KUKA KRL program: MyProgram_112().src

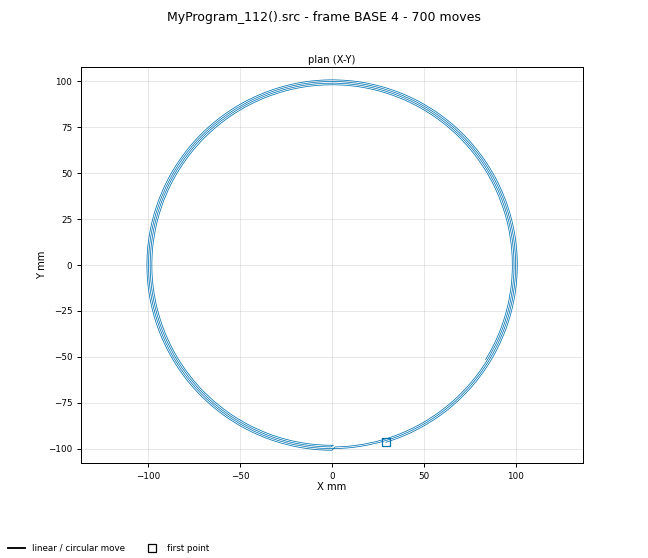
[picture p0: tool path of MyProgram_112().src in frame BASE 4, 700 of 700 moves have a stored position in this frame; points joined in program order, loops and branches not executed]
&ACCESS RVP
&REL 1
&PARAM TEMPLATE = C:\KRC\Roboter\Template\vorgabe
&PARAM EDITMASK = *
DEF MyProgram_112()
; ---- Setting reference (Base) ----
$BASE = BASE_DATA[4]

; --------------------------
; ---- Setting tool (TCP) ----
$TOOL = TOOL_DATA[3]
; --------------------------

$VEL.CP = VEL_APROX_PRINT
Startdeposition()
$VEL.CP = VEL_PRINT
LIN {X 29.2721,Y -96.4972,Z 98,A -76.9707,B 24.9412,C -1.7725,E1 25.0477,E2 162.427} C_DIS
LIN {X 31.6614,Y -95.7396,Z 98,A -75.5501,B 24.941,C -1.7741,E1 25.0514,E2 161.0052} C_DIS
LIN {X 34.0983,Y -94.8985,Z 98,A -74.1594,B 24.941,C -1.7731,E1 25.0551,E2 159.6197} C_DIS
LIN {X 36.321,Y -94.0708,Z 98,A -72.7622,B 24.9408,C -1.7768,E1 25.0587,E2 158.2167} C_DIS
LIN {X 38.5895,Y -93.1634,Z 98,A -71.3458,B 24.9406,C -1.7799,E1 25.0624,E2 156.7962} C_DIS
LIN {X 40.8931,Y -92.1753,Z 98,A -69.8287,B 24.9402,C -1.7857,E1 25.0663,E2 155.269} C_DIS
LIN {X 43.7262,Y -90.8637,Z 98,A -68.0842,B 24.9402,C -1.7874,E1 25.0707,E2 153.525} C_DIS
LIN {X 46.4684,Y -89.4942,Z 98,A -66.439,B 24.9402,C -1.7865,E1 25.0748,E2 151.8866} C_DIS
LIN {X 48.6507,Y -88.3269,Z 98,A -65.038,B 24.94,C -1.7887,E1 25.0782,E2 150.4844} C_DIS
LIN {X 50.7765,Y -87.1224,Z 98,A -63.6258,B 24.9398,C -1.7922,E1 25.0817,E2 149.0682} C_DIS
LIN {X 52.9261,Y -85.8333,Z 98,A -62.2366,B 24.9398,C -1.7935,E1 25.085,E2 147.6803} C_DIS
LIN {X 54.9902,Y -84.526,Z 98,A -60.7105,B 24.9392,C -1.8017,E1 25.0886,E2 146.1398} C_DIS
LIN {X 57.048,Y -83.151,Z 98,A -59.4381,B 24.9393,C -1.7991,E1 25.0915,E2 144.8777} C_DIS
LIN {X 59.0714,Y -81.7259,Z 98,A -57.9396,B 24.9389,C -1.8057,E1 25.0949,E2 143.3689} C_DIS
LIN {X 61.0593,Y -80.2516,Z 98,A -56.6545,B 24.939,C -1.8038,E1 25.0978,E2 142.0928} C_DIS
LIN {X 63.0104,Y -78.729,Z 98,A -55.2547,B 24.9388,C -1.8066,E1 25.1009,E2 140.6917} C_DIS
LIN {X 64.9235,Y -77.1589,Z 98,A -53.7285,B 24.9383,C -1.8146,E1 25.1042,E2 139.1525} C_DIS
LIN {X 66.8211,Y -75.5213,Z 98,A -52.4544,B 24.9385,C -1.8118,E1 25.1068,E2 137.8899} C_DIS
LIN {X 68.6313,Y -73.8803,Z 98,A -51.041,B 24.9382,C -1.8161,E1 25.1097,E2 136.4722} C_DIS
LIN {X 70.4463,Y -72.1516,Z 98,A -49.6565,B 24.9381,C -1.8179,E1 25.1125,E2 135.0891} C_DIS
LIN {X 72.1738,Y -70.4238,Z 98,A -48.2431,B 24.9378,C -1.8224,E1 25.1153,E2 133.6713} C_DIS
LIN {X 74.0767,Y -68.4173,Z 98,A -46.8469,B 24.938,C -1.8192,E1 25.1179,E2 132.2886} C_DIS
LIN {X 75.5424,Y -66.7975,Z 98,A -45.446,B 24.9373,C -1.8289,E1 25.1206,E2 130.8712} C_DIS
LIN {X 77.1791,Y -64.8992,Z 98,A -44.0458,B 24.9371,C -1.8316,E1 25.1231,E2 129.4709} C_DIS
LIN {X 78.7486,Y -62.9856,Z 98,A -42.6477,B 24.9369,C -1.835,E1 25.1256,E2 128.0713} C_DIS
LIN {X 80.2706,Y -61.034,Z 98,A -41.2495,B 24.9366,C -1.8385,E1 25.1279,E2 126.6716} C_DIS
LIN {X 81.7259,Y -59.0714,Z 98,A -39.8536,B 24.9364,C -1.8426,E1 25.1303,E2 125.2726} C_DIS
LIN {X 83.1687,Y -57.0218,Z 98,A -38.454,B 24.9362,C -1.8455,E1 25.1325,E2 123.873} C_DIS
LIN {X 84.526,Y -54.9902,Z 98,A -37.0742,B 24.9359,C -1.8491,E1 25.1346,E2 122.4917} C_DIS
LIN {X 85.8501,Y -52.8992,Z 98,A -35.6606,B 24.9356,C -1.8534,E1 25.1367,E2 121.0751} C_DIS
LIN {X 87.1224,Y -50.7765,Z 98,A -34.2789,B 24.9354,C -1.8565,E1 25.1387,E2 119.6932} C_DIS
LIN {X 88.3423,Y -48.6231,Z 98,A -32.8817,B 24.9351,C -1.8602,E1 25.1406,E2 118.2945} C_DIS
LIN {X 89.5233,Y -46.4122,Z 98,A -31.3317,B 24.9345,C -1.8696,E1 25.1426,E2 116.7305} C_DIS
LIN {X 90.7517,Y -43.9591,Z 98,A -30.0524,B 24.935,C -1.8628,E1 25.1441,E2 115.474} C_DIS
LIN {X 91.6799,Y -41.9925,Z 98,A -28.6902,B 24.9343,C -1.8717,E1 25.1458,E2 114.0982} C_DIS
LIN {X 92.6951,Y -39.7007,Z 98,A -27.2754,B 24.9341,C -1.8757,E1 25.1473,E2 112.6818} C_DIS
LIN {X 93.6299,Y -37.4434,Z 98,A -25.8803,B 24.9337,C -1.8802,E1 25.1488,E2 111.2837} C_DIS
LIN {X 94.5206,Y -35.1343,Z 98,A -24.4705,B 24.9334,C -1.8847,E1 25.1502,E2 109.8712} C_DIS
LIN {X 95.3544,Y -32.8041,Z 98,A -23.0868,B 24.9332,C -1.8882,E1 25.1515,E2 108.487} C_DIS
LIN {X 96.1401,Y -30.4239,Z 98,A -21.7045,B 24.933,C -1.8909,E1 25.1527,E2 107.106} C_DIS
LIN {X 96.8491,Y -28.0857,Z 98,A -20.3095,B 24.9326,C -1.8956,E1 25.1538,E2 105.708} C_DIS
LIN {X 97.8173,Y -24.5019,Z 98,A -18.2145,B 24.9322,C -1.9017,E1 25.1553,E2 103.6107} C_DIS
LIN {X 98.3891,Y -22.094,Z 98,A -16.8179,B 24.9319,C -1.9058,E1 25.1561,E2 102.2126} C_DIS
LIN {X 98.9077,Y -19.6417,Z 98,A -15.4202,B 24.9317,C -1.9092,E1 25.1569,E2 100.8148} C_DIS
LIN {X 99.3547,Y -17.2397,Z 98,A -14.009,B 24.9313,C -1.9146,E1 25.1576,E2 99.3992} C_DIS
LIN {X 99.7479,Y -14.7962,Z 98,A -12.4664,B 24.9305,C -1.9248,E1 25.1583,E2 97.8418} C_DIS
LIN {X 100.2282,Y -11.0833,Z 98,A -10.516,B 24.9305,C -1.9244,E1 25.1589,E2 95.9039} C_DIS
LIN {X 100.47,Y -8.6202,Z 98,A -9.1359,B 24.9303,C -1.9278,E1 25.1593,E2 94.5238} C_DIS
LIN {X 100.6495,Y -6.1835,Z 98,A -7.7249,B 24.9299,C -1.9332,E1 25.1595,E2 93.1083} C_DIS
LIN {X 100.7719,Y -3.68,Z 98,A -6.3269,B 24.9297,C -1.9368,E1 25.1597,E2 91.7103} C_DIS
LIN {X 100.833,Y -1.0408,Z 98,A -4.8838,B 24.9295,C -1.9393,E1 25.1597,E2 90.2699} C_DIS
LIN {X 100.8317,Y 1.2374,Z 98,A -3.5517,B 24.9291,C -1.945,E1 25.1597,E2 88.9323} C_DIS
LIN {X 100.7178,Y 4.9479,Z 98,A -1.4406,B 24.9286,C -1.9518,E1 25.1595,E2 86.8176} C_DIS
LIN {X 100.5661,Y 7.4182,Z 98,A -0.0444,B 24.9283,C -1.9559,E1 25.1593,E2 85.42} C_DIS
LIN {X 100.3193,Y 10.2126,Z 98,A 1.3731,B 24.9284,C -1.9538,E1 25.1589,E2 84.0159} C_DIS
LIN {X 100.0809,Y 12.3438,Z 98,A 2.749,B 24.9277,C -1.9641,E1 25.1585,E2 82.6238} C_DIS
LIN {X 99.743,Y 14.8274,Z 98,A 4.1309,B 24.9275,C -1.9669,E1 25.1579,E2 81.2435} C_DIS
LIN {X 99.3239,Y 17.4113,Z 98,A 5.759,B 24.9267,C -1.9773,E1 25.1571,E2 79.6004} C_DIS
LIN {X 98.7221,Y 20.5475,Z 98,A 7.481,B 24.9266,C -1.9792,E1 25.1562,E2 77.884} C_DIS
LIN {X 98.1031,Y 23.3304,Z 98,A 9.0196,B 24.9264,C -1.9809,E1 25.1552,E2 76.3504} C_DIS
LIN {X 97.501,Y 25.731,Z 98,A 10.4326,B 24.9261,C -1.9855,E1 25.1543,E2 74.9346} C_DIS
LIN {X 96.8491,Y 28.0857,Z 98,A 11.9161,B 24.9255,C -1.9936,E1 25.1531,E2 73.4406} C_DIS
LIN {X 96.0806,Y 30.6089,Z 98,A 13.2351,B 24.9257,C -1.9908,E1 25.152,E2 72.1357} C_DIS
LIN {X 95.3544,Y 32.8041,Z 98,A 14.6225,B 24.9252,C -1.9977,E1 25.1508,E2 70.7398} C_DIS
LIN {X 94.5094,Y 35.1638,Z 98,A 16.0209,B 24.9249,C -2.0008,E1 25.1494,E2 69.3418} C_DIS
LIN {X 93.4675,Y 37.8423,Z 98,A 17.4449,B 24.9252,C -1.9972,E1 25.148,E2 67.9342} C_DIS
LIN {X 92.6702,Y 39.7589,Z 98,A 18.7998,B 24.9244,C -2.0076,E1 25.1465,E2 66.5621} C_DIS
LIN {X 91.6665,Y 42.0211,Z 98,A 20.2138,B 24.9241,C -2.012,E1 25.1449,E2 65.1456} C_DIS
LIN {X 90.6217,Y 44.2297,Z 98,A 21.7975,B 24.9232,C -2.0238,E1 25.1429,E2 63.5425} C_DIS
LIN {X 88.9323,Y 47.5353,Z 98,A 23.6902,B 24.9234,C -2.0208,E1 25.1405,E2 61.6667} C_DIS
LIN {X 87.7232,Y 49.7309,Z 98,A 25.27,B 24.9227,C -2.031,E1 25.1383,E2 60.0712} C_DIS
LIN {X 85.8333,Y 52.9261,Z 98,A 27.2035,B 24.9227,C -2.0295,E1 25.1356,E2 58.1511} C_DIS
LIN {X 84.5086,Y 55.0166,Z 98,A 28.585,B 24.9226,C -2.0322,E1 25.1335,E2 56.7702} C_DIS
LIN {X 83.151,Y 57.048,Z 98,A 29.9824,B 24.9223,C -2.0361,E1 25.1313,E2 55.3705} C_DIS
LIN {X 81.7259,Y 59.0714,Z 98,A 31.3809,B 24.922,C -2.0393,E1 25.129,E2 53.9713} C_DIS
LIN {X 80.2323,Y 61.0843,Z 98,A 32.781,B 24.9218,C -2.0418,E1 25.1267,E2 52.5718} C_DIS
LIN {X 78.729,Y 63.0104,Z 98,A 34.1786,B 24.9215,C -2.0455,E1 25.1242,E2 51.1721} C_DIS
LIN {X 77.1384,Y 64.9476,Z 98,A 35.6387,B 24.9212,C -2.0503,E1 25.1216,E2 49.7074} C_DIS
LIN {X 75.5424,Y 66.7975,Z 98,A 36.9774,B 24.9211,C -2.0515,E1 25.1192,E2 48.3719} C_DIS
LIN {X 73.8587,Y 68.6543,Z 98,A 38.3941,B 24.9209,C -2.0544,E1 25.1165,E2 46.9546} C_DIS
LIN {X 72.1516,Y 70.4463,Z 98,A 39.7773,B 24.9207,C -2.0565,E1 25.1138,E2 45.5723} C_DIS
LIN {X 70.401,Y 72.1957,Z 98,A 41.1938,B 24.9204,C -2.0599,E1 25.111,E2 44.1537} C_DIS
LIN {X 68.2383,Y 74.2409,Z 98,A 42.8629,B 24.9202,C -2.0625,E1 25.1076,E2 42.4853} C_DIS
LIN {X 65.8414,Y 76.3769,Z 98,A 44.7266,B 24.9198,C -2.0677,E1 25.1037,E2 40.6168} C_DIS
LIN {X 63.9472,Y 77.9697,Z 98,A 46.0779,B 24.9198,C -2.0682,E1 25.1008,E2 39.2695} C_DIS
LIN {X 62.0395,Y 79.4963,Z 98,A 47.493,B 24.9195,C -2.0718,E1 25.0977,E2 37.8511} C_DIS
LIN {X 60.0699,Y 80.9949,Z 98,A 48.8783,B 24.9194,C -2.0734,E1 25.0946,E2 36.4669} C_DIS
LIN {X 58.0641,Y 82.4447,Z 98,A 50.2792,B 24.9192,C -2.0756,E1 25.0914,E2 35.0657} C_DIS
LIN {X 56.0233,Y 83.8448,Z 98,A 51.6803,B 24.919,C -2.0777,E1 25.0881,E2 33.6643} C_DIS
LIN {X 53.9488,Y 85.1944,Z 98,A 53.0977,B 24.9188,C -2.0804,E1 25.0848,E2 32.2452} C_DIS
LIN {X 51.5639,Y 86.657,Z 98,A 54.5198,B 24.9192,C -2.0763,E1 25.0814,E2 30.8373} C_DIS
LIN {X 49.6759,Y 87.7544,Z 98,A 55.9032,B 24.9186,C -2.0836,E1 25.0781,E2 29.4408} C_DIS
LIN {X 47.5073,Y 88.947,Z 98,A 57.289,B 24.9186,C -2.0847,E1 25.0747,E2 28.0563} C_DIS
LIN {X 45.1019,Y 90.1894,Z 98,A 58.8834,B 24.9182,C -2.0888,E1 25.0707,E2 26.4565} C_DIS
LIN {X 41.9636,Y 91.6928,Z 98,A 60.795,B 24.9182,C -2.0886,E1 25.0659,E2 24.5503} C_DIS
LIN {X 39.7299,Y 92.6828,Z 98,A 62.1964,B 24.918,C -2.0907,E1 25.0623,E2 23.1475} C_DIS
LIN {X 37.4434,Y 93.6299,Z 98,A 63.618,B 24.9179,C -2.0927,E1 25.0586,E2 21.7243} C_DIS
LIN {X 33.9717,Y 94.9446,Z 98,A 65.7047,B 24.9178,C -2.0938,E1 25.0531,E2 19.6394} C_DIS
LIN {X 31.3215,Y 95.85,Z 98,A 67.1448,B 24.9181,C -2.0894,E1 25.0494,E2 18.2124} C_DIS
LIN {X 28.9746,Y 96.5854,Z 98,A 68.7109,B 24.9175,C -2.0969,E1 25.0451,E2 16.6315} C_DIS
LIN {X 25.6699,Y 97.5171,Z 98,A 70.6199,B 24.9175,C -2.0966,E1 25.04,E2 14.7264} C_DIS
LIN {X 23.2997,Y 98.1106,Z 98,A 72.0231,B 24.9175,C -2.0979,E1 25.0362,E2 13.322} C_DIS
LIN {X 20.854,Y 98.6592,Z 98,A 73.4458,B 24.9175,C -2.0986,E1 25.0323,E2 11.8996} C_DIS
LIN {X 18.4576,Y 99.1357,Z 98,A 74.8488,B 24.9173,C -2.0997,E1 25.0285,E2 10.4955} C_DIS
LIN {X 15.9879,Y 99.5636,Z 98,A 76.2394,B 24.9173,C -2.0989,E1 25.0246,E2 9.1082} C_DIS
LIN {X 13.5397,Y 99.926,Z 98,A 77.6611,B 24.9173,C -2.0999,E1 25.0207,E2 7.6855} C_DIS
LIN {X 11.0833,Y 100.2282,Z 98,A 79.0669,B 24.9173,C -2.1001,E1 25.0168,E2 6.2802} C_DIS
LIN {X 8.2393,Y 100.5004,Z 98,A 80.4739,B 24.9179,C -2.0922,E1 25.013,E2 4.8927} C_DIS
LIN {X 6.1835,Y 100.6495,Z 98,A 81.8774,B 24.9172,C -2.1009,E1 25.009,E2 3.4694} C_DIS
LIN {X 3.68,Y 100.7719,Z 98,A 83.3917,B 24.917,C -2.1041,E1 25.0047,E2 1.9478} C_DIS
LIN {X 1.2375,Y 100.8317,Z 98,A 84.6904,B 24.9172,C -2.1006,E1 25.0011,E2 0.6576} C_DIS
LIN {X -1.2375,Y 100.8317,Z 98,A 86.155,B 24.9172,C -2.1025,E1 24.997,E2 -0.8114} C_DIS
LIN {X -3.7432,Y 100.7696,Z 98,A 87.4895,B 24.9174,C -2.0987,E1 24.9933,E2 -2.1373} C_DIS
LIN {X -6.2151,Y 100.6474,Z 98,A 88.8969,B 24.9174,C -2.0982,E1 24.9894,E2 -3.5439} C_DIS
LIN {X -8.7058,Y 100.4624,Z 98,A 90.4498,B 24.9171,C -2.1025,E1 24.9851,E2 -5.1076} C_DIS
LIN {X -11.1147,Y 100.2249,Z 98,A 91.7112,B 24.9175,C -2.0976,E1 24.9816,E2 -6.3581} C_DIS
LIN {X -13.8731,Y 99.879,Z 98,A 93.327,B 24.9175,C -2.098,E1 24.9771,E2 -7.976} C_DIS
LIN {X -17.2708,Y 99.3491,Z 98,A 95.2333,B 24.9177,C -2.0948,E1 24.9719,E2 -9.8766} C_DIS
LIN {X -19.7037,Y 98.8953,Z 98,A 96.8487,B 24.9172,C -2.1013,E1 24.9674,E2 -11.5092} C_DIS
LIN {X -23.3304,Y 98.1031,Z 98,A 98.7557,B 24.9179,C -2.0921,E1 24.9623,E2 -13.3967} C_DIS
LIN {X -25.731,Y 97.501,Z 98,A 100.1813,B 24.9179,C -2.0914,E1 24.9584,E2 -14.8227} C_DIS
LIN {X -28.116,Y 96.8401,Z 98,A 101.5743,B 24.9181,C -2.0894,E1 24.9547,E2 -16.2133} C_DIS
LIN {X -30.4541,Y 96.1307,Z 98,A 102.999,B 24.9181,C -2.0891,E1 24.9509,E2 -17.6398} C_DIS
LIN {X -32.8339,Y 95.3439,Z 98,A 104.4107,B 24.9183,C -2.087,E1 24.9471,E2 -19.0491} C_DIS
LIN {X -35.1343,Y 94.5206,Z 98,A 105.9422,B 24.9181,C -2.0903,E1 24.9431,E2 -20.5916} C_DIS
LIN {X -37.4434,Y 93.6299,Z 98,A 107.2295,B 24.9185,C -2.0841,E1 24.9398,E2 -21.867} C_DIS
LIN {X -39.7589,Y 92.6702,Z 98,A 108.6255,B 24.9188,C -2.0811,E1 24.9362,E2 -23.2589} C_DIS
LIN {X -41.9925,Y 91.6799,Z 98,A 110.0512,B 24.9188,C -2.0803,E1 24.9326,E2 -24.6863} C_DIS
LIN {X -44.2581,Y 90.6077,Z 98,A 111.5825,B 24.9188,C -2.0819,E1 24.9287,E2 -26.2253} C_DIS
LIN {X -46.4404,Y 89.5089,Z 98,A 112.8732,B 24.9192,C -2.0761,E1 24.9255,E2 -27.5058} C_DIS
LIN {X -48.6231,Y 88.3423,Z 98,A 114.2848,B 24.9193,C -2.0739,E1 24.9221,E2 -28.9163} C_DIS
LIN {X -50.7765,Y 87.1224,Z 98,A 115.6806,B 24.9196,C -2.0711,E1 24.9187,E2 -30.3094} C_DIS
LIN {X -52.8993,Y 85.8501,Z 98,A 117.2564,B 24.9193,C -2.0745,E1 24.9149,E2 -31.8982} C_DIS
LIN {X -55.6124,Y 84.1157,Z 98,A 119.0031,B 24.9198,C -2.0681,E1 24.9108,E2 -33.6352} C_DIS
LIN {X -58.0641,Y 82.4447,Z 98,A 120.6229,B 24.9202,C -2.0624,E1 24.9071,E2 -35.2469} C_DIS
LIN {X -60.0699,Y 80.9949,Z 98,A 122.0517,B 24.9204,C -2.0603,E1 24.9039,E2 -36.6758} C_DIS
LIN {X -62.0395,Y 79.4963,Z 98,A 123.4485,B 24.9207,C -2.0569,E1 24.9008,E2 -38.0698} C_DIS
LIN {X -63.9718,Y 77.9498,Z 98,A 124.8613,B 24.9209,C -2.0541,E1 24.8978,E2 -39.4811} C_DIS
LIN {X -65.8893,Y 76.3356,Z 98,A 126.2927,B 24.9211,C -2.0512,E1 24.8947,E2 -40.9111} C_DIS
LIN {X -67.7195,Y 74.717,Z 98,A 127.6877,B 24.9213,C -2.0482,E1 24.8918,E2 -42.3046} C_DIS
LIN {X -69.5328,Y 73.0326,Z 98,A 129.2763,B 24.9211,C -2.0513,E1 24.8886,E2 -43.9071} C_DIS
LIN {X -72.1738,Y 70.4238,Z 98,A 131.2381,B 24.9219,C -2.0411,E1 24.8847,E2 -45.8528} C_DIS
LIN {X -73.9017,Y 68.608,Z 98,A 132.6372,B 24.9222,C -2.0367,E1 24.8821,E2 -47.2475} C_DIS
LIN {X -75.5632,Y 66.7737,Z 98,A 134.0677,B 24.9224,C -2.0339,E1 24.8794,E2 -48.6779} C_DIS
LIN {X -77.1791,Y 64.8992,Z 98,A 135.4821,B 24.9227,C -2.0306,E1 24.8769,E2 -50.0908} C_DIS
LIN {X -78.7486,Y 62.9856,Z 98,A 136.8963,B 24.9229,C -2.0272,E1 24.8744,E2 -51.5035} C_DIS
LIN {X -80.4938,Y 60.7369,Z 98,A 138.3351,B 24.9237,C -2.0167,E1 24.872,E2 -52.9243} C_DIS
LIN {X -81.7259,Y 59.0714,Z 98,A 139.7235,B 24.9234,C -2.0208,E1 24.8696,E2 -54.329} C_DIS
LIN {X -83.1687,Y 57.0218,Z 98,A 141.1235,B 24.9238,C -2.016,E1 24.8674,E2 -55.7245} C_DIS
LIN {X -84.526,Y 54.9902,Z 98,A 142.5369,B 24.924,C -2.013,E1 24.8652,E2 -57.1378} C_DIS
LIN {X -86.0619,Y 52.5507,Z 98,A 143.9946,B 24.9248,C -2.0022,E1 24.8631,E2 -58.5773} C_DIS
LIN {X -87.1224,Y 50.7765,Z 98,A 145.3834,B 24.9245,C -2.0062,E1 24.8611,E2 -59.9827} C_DIS
LIN {X -88.3574,Y 48.5953,Z 98,A 146.8002,B 24.9249,C -2.0018,E1 24.8592,E2 -61.3964} C_DIS
LIN {X -89.5233,Y 46.4122,Z 98,A 148.2158,B 24.9252,C -1.998,E1 24.8574,E2 -62.8104} C_DIS
LIN {X -91.1576,Y 43.1144,Z 98,A 150.337,B 24.9255,C -1.9927,E1 24.8548,E2 -64.9307} C_DIS
LIN {X -92.1883,Y 40.8642,Z 98,A 151.7364,B 24.9259,C -1.9883,E1 24.8532,E2 -66.3271} C_DIS
LIN {X -93.3228,Y 38.1979,Z 98,A 153.1958,B 24.9267,C -1.9769,E1 24.8516,E2 -67.7675} C_DIS
LIN {X -94.0823,Y 36.2916,Z 98,A 154.7307,B 24.9261,C -1.9859,E1 24.85,E2 -69.3324} C_DIS
LIN {X -94.9446,Y 33.9717,Z 98,A 155.9836,B 24.9268,C -1.9763,E1 24.8488,E2 -70.5695} C_DIS
LIN {X -95.8212,Y 31.4107,Z 98,A 157.4296,B 24.9274,C -1.9684,E1 24.8476,E2 -72.0049} C_DIS
LIN {X -96.4972,Y 29.2721,Z 98,A 158.8317,B 24.9274,C -1.9687,E1 24.8464,E2 -73.4159} C_DIS
LIN {X -97.1865,Y 26.8951,Z 98,A 160.2475,B 24.9276,C -1.9646,E1 24.8453,E2 -74.8301} C_DIS
LIN {X -98.1106,Y 23.2997,Z 98,A 162.3553,B 24.9281,C -1.9579,E1 24.8439,E2 -76.9342} C_DIS
LIN {X -98.704,Y 20.6355,Z 98,A 163.8036,B 24.9287,C -1.9495,E1 24.843,E2 -78.3709} C_DIS
LIN {X -99.1357,Y 18.4576,Z 98,A 165.2037,B 24.9287,C -1.9501,E1 24.8423,E2 -79.7809} C_DIS
LIN {X -99.5588,Y 16.0191,Z 98,A 166.6035,B 24.929,C -1.9454,E1 24.8417,E2 -81.1777} C_DIS
LIN {X -100.0809,Y 12.3438,Z 98,A 168.7441,B 24.9295,C -1.9397,E1 24.8409,E2 -83.3175} C_DIS
LIN {X -100.3537,Y 9.884,Z 98,A 170.1603,B 24.9298,C -1.9355,E1 24.8405,E2 -84.7321} C_DIS
LIN {X -100.5661,Y 7.4182,Z 98,A 171.5766,B 24.9301,C -1.9313,E1 24.8401,E2 -86.1469} C_DIS
LIN {X -100.7178,Y 4.9479,Z 98,A 173.1612,B 24.93,C -1.9329,E1 24.8399,E2 -87.7448} C_DIS
LIN {X -100.8095,Y 2.4431,Z 98,A 174.4805,B 24.9305,C -1.9247,E1 24.8399,E2 -89.0526} C_DIS
LIN {X -100.8387,Y 0,Z 98,A 175.7839,B 24.9311,C -1.9174,E1 24.8398,E2 -90.3462} C_DIS
LIN {X -100.8052,Y -2.595,Z 98,A 177.2307,B 24.9315,C -1.9117,E1 24.8398,E2 -91.7883} C_DIS
LIN {X -100.7161,Y -4.9795,Z 98,A 178.6591,B 24.9316,C -1.9098,E1 24.84,E2 -93.2207} C_DIS
LIN {X -100.5661,Y -7.4182,Z 98,A -179.9426,B 24.9319,C -1.9057,E1 24.8403,E2 -94.6177} C_DIS
LIN {X -100.3537,Y -9.884,Z 98,A -178.5105,B 24.9322,C -1.9021,E1 24.8407,E2 -96.0498} C_DIS
LIN {X -100.0809,Y -12.3438,Z 98,A -177.0942,B 24.9325,C -1.898,E1 24.8411,E2 -97.4648} C_DIS
LIN {X -99.7479,Y -14.7962,Z 98,A -175.6786,B 24.9328,C -1.8939,E1 24.8417,E2 -98.8791} C_DIS
LIN {X -99.3491,Y -17.2708,Z 98,A -174.2775,B 24.9331,C -1.8886,E1 24.8423,E2 -100.2759} C_DIS
LIN {X -98.8953,Y -19.7037,Z 98,A -172.8448,B 24.9334,C -1.8852,E1 24.8431,E2 -101.7088} C_DIS
LIN {X -98.382,Y -22.1248,Z 98,A -171.4293,B 24.9337,C -1.8811,E1 24.8439,E2 -103.123} C_DIS
LIN {X -97.8173,Y -24.5019,Z 98,A -170.0152,B 24.9339,C -1.8777,E1 24.8449,E2 -104.5373} C_DIS
LIN {X -97.1779,Y -26.9255,Z 98,A -168.5975,B 24.9342,C -1.8732,E1 24.8459,E2 -105.9524} C_DIS
LIN {X -96.4972,Y -29.2721,Z 98,A -167.2003,B 24.9345,C -1.8693,E1 24.847,E2 -107.3483} C_DIS
LIN {X -95.7396,Y -31.6614,Z 98,A -165.7666,B 24.9348,C -1.8654,E1 24.8483,E2 -108.7809} C_DIS
LIN {X -94.9338,Y -34.0014,Z 98,A -164.3679,B 24.9351,C -1.8609,E1 24.8495,E2 -110.177} C_DIS
LIN {X -94.0708,Y -36.321,Z 98,A -162.9527,B 24.9353,C -1.8571,E1 24.8509,E2 -111.5911} C_DIS
LIN {X -93.1634,Y -38.5895,Z 98,A -161.5228,B 24.9355,C -1.8545,E1 24.8525,E2 -113.0228} C_DIS
LIN {X -92.1753,Y -40.8931,Z 98,A -160.1224,B 24.9359,C -1.8497,E1 24.854,E2 -114.4193} C_DIS
LIN {X -91.1439,Y -43.1428,Z 98,A -158.6648,B 24.936,C -1.8475,E1 24.8557,E2 -115.8795} C_DIS
LIN {X -90.0721,Y -45.3385,Z 98,A -157.2777,B 24.9363,C -1.8436,E1 24.8575,E2 -117.2648} C_DIS
LIN {X -88.8054,Y -47.7692,Z 98,A -155.8466,B 24.9369,C -1.8349,E1 24.8593,E2 -118.6829} C_DIS
LIN {X -87.7232,Y -49.7309,Z 98,A -154.4634,B 24.9369,C -1.8353,E1 24.8612,E2 -120.0743} C_DIS
LIN {X -86.4763,Y -51.8688,Z 98,A -153.0322,B 24.9371,C -1.8324,E1 24.8632,E2 -121.506} C_DIS
LIN {X -85.1774,Y -53.9754,Z 98,A -151.6346,B 24.9373,C -1.8285,E1 24.8653,E2 -122.9013} C_DIS
LIN {X -83.8448,Y -56.0233,Z 98,A -150.0781,B 24.9372,C -1.8308,E1 24.8677,E2 -124.4712} C_DIS
LIN {X -82.4263,Y -58.0898,Z 98,A -148.8065,B 24.9378,C -1.8219,E1 24.8697,E2 -125.7277} C_DIS
LIN {X -80.9949,Y -60.0699,Z 98,A -147.2553,B 24.9376,C -1.8242,E1 24.8723,E2 -127.2919} C_DIS
LIN {X -79.4963,Y -62.0395,Z 98,A -145.9803,B 24.9382,C -1.8162,E1 24.8745,E2 -128.5539} C_DIS
LIN {X -77.9498,Y -63.9718,Z 98,A -144.3875,B 24.938,C -1.8194,E1 24.8773,E2 -130.1618} C_DIS
LIN {X -76.3356,Y -65.8893,Z 98,A -143.1355,B 24.9386,C -1.8101,E1 24.8796,E2 -131.3973} C_DIS
LIN {X -74.5425,Y -67.9097,Z 98,A -141.7283,B 24.9391,C -1.8021,E1 24.8822,E2 -132.7919} C_DIS
LIN {X -72.7676,Y -69.8077,Z 98,A -140.2864,B 24.9394,C -1.7977,E1 24.8849,E2 -134.2294} C_DIS
LIN {X -70.4238,Y -72.1738,Z 98,A -138.1919,B 24.9392,C -1.8008,E1 24.8891,E2 -136.3402} C_DIS
LIN {X -68.608,Y -73.9017,Z 98,A -136.7941,B 24.9395,C -1.797,E1 24.8919,E2 -137.7346} C_DIS
LIN {X -66.7975,Y -75.5424,Z 98,A -135.3671,B 24.9395,C -1.7956,E1 24.8949,E2 -139.1641} C_DIS
LIN {X -64.8992,Y -77.1791,Z 98,A -133.9092,B 24.9397,C -1.7941,E1 24.898,E2 -140.624} C_DIS
LIN {X -62.9856,Y -78.7486,Z 98,A -132.5412,B 24.9399,C -1.7901,E1 24.901,E2 -141.9877} C_DIS
LIN {X -60.7463,Y -80.4868,Z 98,A -131.1058,B 24.9405,C -1.781,E1 24.9041,E2 -143.4066} C_DIS
LIN {X -59.0714,Y -81.7259,Z 98,A -129.5443,B 24.9398,C -1.7925,E1 24.9077,E2 -145.001} C_DIS
LIN {X -55.9969,Y -83.8622,Z 98,A -127.6174,B 24.9405,C -1.7818,E1 24.9121,E2 -146.9089} C_DIS
LIN {X -53.9488,Y -85.1944,Z 98,A -126.1066,B 24.9403,C -1.7841,E1 24.9157,E2 -148.43} C_DIS
LIN {X -51.8145,Y -86.5088,Z 98,A -124.796,B 24.9408,C -1.7779,E1 24.9188,E2 -149.7299} C_DIS
LIN {X -49.7035,Y -87.739,Z 98,A -123.3868,B 24.9408,C -1.7767,E1 24.9222,E2 -151.1404} C_DIS
LIN {X -46.4122,Y -89.5233,Z 98,A -121.1498,B 24.9408,C -1.7779,E1 24.9277,E2 -153.3866} C_DIS
LIN {X -44.2298,Y -90.6217,Z 98,A -119.8453,B 24.9411,C -1.7731,E1 24.931,E2 -154.6832} C_DIS
LIN {X -41.9925,Y -91.6799,Z 98,A -118.4516,B 24.9412,C -1.7711,E1 24.9345,E2 -156.0755} C_DIS
LIN {X -39.7007,Y -92.6951,Z 98,A -117.0241,B 24.9413,C -1.7697,E1 24.9382,E2 -157.503} C_DIS
LIN {X -37.4434,Y -93.6299,Z 98,A -115.6165,B 24.9413,C -1.769,E1 24.9418,E2 -158.9121} C_DIS
LIN {X -35.1343,Y -94.5206,Z 98,A -114.2237,B 24.9415,C -1.7672,E1 24.9454,E2 -160.3035} C_DIS
LIN {X -32.8041,Y -95.3544,Z 98,A -112.7987,B 24.9415,C -1.7667,E1 24.9492,E2 -161.7301} C_DIS
LIN {X -30.4239,Y -96.1401,Z 98,A -111.4046,B 24.9416,C -1.7645,E1 24.9529,E2 -163.1215} C_DIS
LIN {X -28.0857,Y -96.8491,Z 98,A -109.9979,B 24.9416,C -1.7642,E1 24.9567,E2 -164.5299} C_DIS
LIN {X -25.6699,Y -97.5171,Z 98,A -108.5882,B 24.9418,C -1.7628,E1 24.9605,E2 -165.9383} C_DIS
LIN {X -23.2997,Y -98.1106,Z 98,A -107.0541,B 24.9414,C -1.7675,E1 24.9647,E2 -167.4857} C_DIS
LIN {X -20.885,Y -98.6528,Z 98,A -105.758,B 24.9418,C -1.7627,E1 24.9682,E2 -168.7722} C_DIS
LIN {X -18.4576,Y -99.1357,Z 98,A -104.3666,B 24.9418,C -1.7616,E1 24.972,E2 -170.1624} C_DIS
LIN {X -15.9879,Y -99.5636,Z 98,A -102.958,B 24.9419,C -1.7606,E1 24.9759,E2 -171.57} C_DIS
LIN {X -13.5397,Y -99.926,Z 98,A -101.4416,B 24.9417,C -1.7645,E1 24.9801,E2 -173.0967} C_DIS
LIN {X -10.4565,Y -100.2938,Z 98,A -99.6599,B 24.9417,C -1.7649,E1 24.985,E2 -174.8806} C_DIS
LIN {X -7.4182,Y -100.5661,Z 98,A -98.0362,B 24.9419,C -1.7607,E1 24.9895,E2 -176.495} C_DIS
LIN {X -4.9164,Y -100.7192,Z 98,A -96.6124,B 24.9419,C -1.7607,E1 24.9935,E2 -177.9194} C_DIS
LIN {X -2.4431,Y -100.8095,Z 98,A -95.2229,B 24.9419,C -1.7603,E1 24.9974,E2 -179.3081} C_DIS
LIN {X 0.0316,Y -100.8391,Z 98,A -93.8175,B 24.9419,C -1.7606,E1 25.0013,E2 -180.714} C_DIS
LIN {X 0.0316,Y -100.8391,Z 98,A -93.8175,B 24.9419,C -1.7606,E1 25.0013,E2 -180.714} C_DIS
Enddeposition()
LIN {X 0.6838,Y -99.9382,Z 98,A -93.4786,B 24.9409,C -1.775,E1 25.0023,E2 -181.0872} C_DIS
Startdeposition()
$VEL.CP = VEL_PRINT
LIN {X -2.9468,Y -99.8985,Z 98,A -96.3512,B 24.9429,C -1.7451,E1 24.9941,E2 -178.1434} C_DIS
LIN {X -6.3381,Y -99.7416,Z 98,A -98.2134,B 24.9427,C -1.748,E1 24.9889,E2 -176.2877} C_DIS
LIN {X -11.0042,Y -99.3361,Z 98,A -100.8162,B 24.9425,C -1.7512,E1 24.9817,E2 -173.6912} C_DIS
LIN {X -13.6034,Y -99.0128,Z 98,A -102.7533,B 24.9435,C -1.7356,E1 24.9763,E2 -171.7156} C_DIS
LIN {X -20.6975,Y -97.7771,Z 98,A -106.4496,B 24.9424,C -1.7528,E1 24.9662,E2 -168.0562} C_DIS
LIN {X -23.2449,Y -97.2011,Z 98,A -108.4598,B 24.9436,C -1.735,E1 24.9606,E2 -166.001} C_DIS
LIN {X -29.56,Y -95.4704,Z 98,A -111.6895,B 24.9422,C -1.7564,E1 24.9521,E2 -162.817} C_DIS
LIN {X -32.4539,Y -94.5274,Z 98,A -113.4544,B 24.9422,C -1.7571,E1 24.9474,E2 -161.0503} C_DIS
LIN {X -34.8997,Y -93.6519,Z 98,A -115.1151,B 24.9425,C -1.7523,E1 24.943,E2 -159.3748} C_DIS
LIN {X -38.0403,Y -92.4201,Z 98,A -117.0289,B 24.9423,C -1.7549,E1 24.9381,E2 -157.4631} C_DIS
LIN {X -41.2058,Y -91.0522,Z 98,A -118.9328,B 24.942,C -1.7597,E1 24.9332,E2 -155.5659} C_DIS
LIN {X -43.7013,Y -89.8821,Z 98,A -120.6412,B 24.9421,C -1.757,E1 24.9289,E2 -153.8468} C_DIS
LIN {X -46.5275,Y -88.451,Z 98,A -122.3824,B 24.9418,C -1.762,E1 24.9246,E2 -152.1127} C_DIS
LIN {X -49.7211,Y -86.6961,Z 98,A -124.2058,B 24.941,C -1.7742,E1 24.9202,E2 -150.3132} C_DIS
LIN {X -51.8877,Y -85.417,Z 98,A -125.9121,B 24.9415,C -1.767,E1 24.916,E2 -148.5845} C_DIS
LIN {X -54.7129,Y -83.6362,Z 98,A -127.7964,B 24.9412,C -1.771,E1 24.9116,E2 -146.7036} C_DIS
LIN {X -57.6116,Y -81.6675,Z 98,A -129.9903,B 24.9414,C -1.7678,E1 24.9065,E2 -144.4947} C_DIS
LIN {X -60.3775,Y -79.6438,Z 98,A -131.9548,B 24.9412,C -1.7712,E1 24.9022,E2 -142.5314} C_DIS
LIN {X -63.7278,Y -76.9882,Z 98,A -134.2985,B 24.9406,C -1.7795,E1 24.8971,E2 -140.1985} C_DIS
LIN {X -66.2396,Y -74.84,Z 98,A -136.3999,B 24.9409,C -1.776,E1 24.8926,E2 -138.0806} C_DIS
LIN {X -68.6438,Y -72.6393,Z 98,A -138.2609,B 24.9406,C -1.7801,E1 24.8888,E2 -136.2216} C_DIS
LIN {X -70.9746,Y -70.3635,Z 98,A -140.0004,B 24.94,C -1.7884,E1 24.8854,E2 -134.4947} C_DIS
LIN {X -73.6757,Y -67.5298,Z 98,A -142.268,B 24.9398,C -1.7926,E1 24.8811,E2 -132.2271} C_DIS
LIN {X -76.4552,Y -64.3683,Z 98,A -144.6012,B 24.9392,C -1.8008,E1 24.8768,E2 -129.903} C_DIS
LIN {X -78.2737,Y -62.1422,Z 98,A -146.2602,B 24.939,C -1.8044,E1 24.8739,E2 -128.2446} C_DIS
LIN {X -80.1241,Y -59.7382,Z 98,A -148.3113,B 24.9394,C -1.798,E1 24.8705,E2 -126.1684} C_DIS
LIN {X -82.301,Y -56.7019,Z 98,A -150.0996,B 24.9382,C -1.8153,E1 24.8676,E2 -124.4127} C_DIS
LIN {X -84.1621,Y -53.8993,Z 98,A -152.0362,B 24.9379,C -1.82,E1 24.8647,E2 -122.4776} C_DIS
LIN {X -86.1362,Y -50.6852,Z 98,A -154.2251,B 24.9376,C -1.8248,E1 24.8615,E2 -120.2889} C_DIS
LIN {X -87.7746,Y -47.7916,Z 98,A -156.6202,B 24.9384,C -1.8135,E1 24.8582,E2 -117.8542} C_DIS
LIN {X -89.2723,Y -44.9357,Z 98,A -158.2294,B 24.9375,C -1.8266,E1 24.8562,E2 -116.2677} C_DIS
LIN {X -90.876,Y -41.5967,Z 98,A -160.119,B 24.9365,C -1.8405,E1 24.854,E2 -114.4009} C_DIS
LIN {X -92.1878,Y -38.5987,Z 98,A -162.0114,B 24.9362,C -1.8454,E1 24.8519,E2 -112.5095} C_DIS
LIN {X -93.7469,Y -34.6421,Z 98,A -164.3552,B 24.9355,C -1.8556,E1 24.8496,E2 -110.1771} C_DIS
LIN {X -95.6488,Y -28.9832,Z 98,A -168.0961,B 24.9355,C -1.8551,E1 24.8463,E2 -106.4136} C_DIS
LIN {X -96.4757,Y -26.0927,Z 98,A -169.5846,B 24.9346,C -1.8683,E1 24.8452,E2 -104.9478} C_DIS
LIN {X -97.2338,Y -23.1152,Z 98,A -171.4086,B 24.9343,C -1.8715,E1 24.8439,E2 -103.1209} C_DIS
LIN {X -97.6889,Y -21.1024,Z 98,A -172.5742,B 24.934,C -1.8758,E1 24.8432,E2 -101.9587} C_DIS
LIN {X -98.3001,Y -18.0444,Z 98,A -174.4536,B 24.9339,C -1.8783,E1 24.8422,E2 -100.0742} C_DIS
LIN {X -98.747,Y -15.4092,Z 98,A -176.0915,B 24.9338,C -1.8796,E1 24.8415,E2 -98.4297} C_DIS
LIN {X -99.1689,Y -12.4138,Z 98,A -177.6738,B 24.933,C -1.8901,E1 24.8409,E2 -96.863} C_DIS
LIN {X -99.4448,Y -9.9657,Z 98,A -179.3384,B 24.9333,C -1.8862,E1 24.8404,E2 -95.1791} C_DIS
LIN {X -99.7462,Y -6.2692,Z 98,A 178.5556,B 24.9328,C -1.8937,E1 24.84,E2 -93.0782} C_DIS
LIN {X -99.9147,Y -2.3983,Z 98,A 176.5372,B 24.9318,C -1.9075,E1 24.8398,E2 -91.0807} C_DIS
LIN {X -99.9393,Y 0.7125,Z 98,A 174.5741,B 24.9318,C -1.9073,E1 24.8398,E2 -89.1052} C_DIS
LIN {X -99.8513,Y 4.2558,Z 98,A 172.5727,B 24.9313,C -1.9149,E1 24.84,E2 -87.1098} C_DIS
LIN {X -99.6273,Y 7.9239,Z 98,A 170.383,B 24.931,C -1.9189,E1 24.8404,E2 -84.9166} C_DIS
LIN {X -99.3441,Y 10.9279,Z 98,A 168.6032,B 24.9307,C -1.9228,E1 24.8409,E2 -83.1354} C_DIS
LIN {X -98.9346,Y 14.154,Z 98,A 166.9192,B 24.9298,C -1.9348,E1 24.8415,E2 -81.47} C_DIS
LIN {X -98.4511,Y 17.2048,Z 98,A 165.2048,B 24.9293,C -1.9423,E1 24.8423,E2 -79.7633} C_DIS
LIN {X -97.9016,Y 20.0916,Z 98,A 163.2966,B 24.9294,C -1.9403,E1 24.8434,E2 -77.839} C_DIS
LIN {X -97.0542,Y 23.8517,Z 98,A 161.0355,B 24.929,C -1.9456,E1 24.8448,E2 -75.5774} C_DIS
LIN {X -96.1714,Y 27.1928,Z 98,A 159.374,B 24.9278,C -1.9625,E1 24.846,E2 -73.9464} C_DIS
LIN {X -95.4228,Y 29.7136,Z 98,A 157.3236,B 24.9288,C -1.9492,E1 24.8477,E2 -71.8526} C_DIS
LIN {X -93.7877,Y 34.5304,Z 98,A 154.5837,B 24.9277,C -1.9641,E1 24.8502,E2 -69.1325} C_DIS
LIN {X -92.5122,Y 37.814,Z 98,A 152.6852,B 24.9269,C -1.9743,E1 24.8522,E2 -67.2478} C_DIS
LIN {X -90.6501,Y 42.0827,Z 98,A 149.9586,B 24.9265,C -1.9805,E1 24.8553,E2 -64.5209} C_DIS
LIN {X -89.3011,Y 44.8777,Z 98,A 148.2633,B 24.9259,C -1.9885,E1 24.8573,E2 -62.8358} C_DIS
LIN {X -88.3309,Y 46.7556,Z 98,A 147.0717,B 24.9255,C -1.9928,E1 24.8589,E2 -61.6479} C_DIS
LIN {X -87.3178,Y 48.621,Z 98,A 145.8603,B 24.9253,C -1.9965,E1 24.8605,E2 -60.4391} C_DIS
LIN {X -86.2572,Y 50.4804,Z 98,A 144.4187,B 24.9255,C -1.9929,E1 24.8625,E2 -58.9813} C_DIS
LIN {X -83.6582,Y 54.679,Z 98,A 141.128,B 24.9261,C -1.9856,E1 24.8675,E2 -55.6564} C_DIS
LIN {X -81.6692,Y 57.6092,Z 98,A 139.16,B 24.9255,C -1.9932,E1 24.8707,E2 -53.697} C_DIS
LIN {X -78.9299,Y 61.3075,Z 98,A 136.986,B 24.9238,C -2.0158,E1 24.8743,E2 -51.5665} C_DIS
LIN {X -76.4839,Y 64.3347,Z 98,A 134.7396,B 24.9234,C -2.0211,E1 24.8782,E2 -49.3223} C_DIS
LIN {X -73.9286,Y 67.2541,Z 98,A 132.4075,B 24.9233,C -2.0231,E1 24.8826,E2 -46.9846} C_DIS
LIN {X -71.5647,Y 69.7653,Z 98,A 130.5732,B 24.9225,C -2.0328,E1 24.8861,E2 -45.1654} C_DIS
LIN {X -69.6748,Y 71.652,Z 98,A 128.841,B 24.9228,C -2.0297,E1 24.8896,E2 -43.4185} C_DIS
LIN {X -66.9778,Y 74.1791,Z 98,A 126.812,B 24.9221,C -2.0376,E1 24.8937,E2 -41.4002} C_DIS
LIN {X -64.6033,Y 76.2553,Z 98,A 125.1677,B 24.9214,C -2.0473,E1 24.8971,E2 -39.7725} C_DIS
LIN {X -62.6925,Y 77.834,Z 98,A 123.5607,B 24.9217,C -2.0441,E1 24.9006,E2 -38.1517} C_DIS
LIN {X -60.0086,Y 79.9209,Z 98,A 121.5913,B 24.9214,C -2.0475,E1 24.905,E2 -36.1833} C_DIS
LIN {X -56.8773,Y 82.1791,Z 98,A 118.9901,B 24.9221,C -2.0387,E1 24.911,E2 -33.5523} C_DIS
LIN {X -52.4181,Y 85.0946,Z 98,A 115.8861,B 24.9218,C -2.0427,E1 24.9184,E2 -30.448} C_DIS
LIN {X -46.1504,Y 88.6496,Z 98,A 112.0261,B 24.9205,C -2.0592,E1 24.9277,E2 -26.6161} C_DIS
LIN {X -43.2522,Y 90.0979,Z 98,A 110.1284,B 24.9204,C -2.0608,E1 24.9325,E2 -24.7171} C_DIS
LIN {X -40.3941,Y 91.4163,Z 98,A 108.3849,B 24.92,C -2.0655,E1 24.9369,E2 -22.9808} C_DIS
LIN {X -37.0001,Y 92.8419,Z 98,A 106.2707,B 24.9198,C -2.0683,E1 24.9424,E2 -20.8686} C_DIS
LIN {X -33.595,Y 94.1278,Z 98,A 104.1532,B 24.9196,C -2.07,E1 24.9479,E2 -18.7506} C_DIS
LIN {X -29.9665,Y 95.3443,Z 98,A 102.0155,B 24.9193,C -2.0745,E1 24.9536,E2 -16.6199} C_DIS
LIN {X -27.3601,Y 96.124,Z 98,A 100.5594,B 24.9189,C -2.0799,E1 24.9575,E2 -15.1742} C_DIS
LIN {X -24.2531,Y 96.9562,Z 98,A 98.7751,B 24.9186,C -2.0838,E1 24.9623,E2 -13.3965} C_DIS
LIN {X -21.6504,Y 97.5693,Z 98,A 97.1257,B 24.9188,C -2.0811,E1 24.9668,E2 -11.7385} C_DIS
LIN {X -19.1083,Y 98.0985,Z 98,A 95.8101,B 24.9182,C -2.0885,E1 24.9703,E2 -10.4389} C_DIS
LIN {X -17.0324,Y 98.4814,Z 98,A 94.5477,B 24.9182,C -2.0875,E1 24.9738,E2 -9.173} C_DIS
LIN {X -9.9297,Y 99.4486,Z 98,A 90.4699,B 24.918,C -2.0911,E1 24.9851,E2 -5.1008} C_DIS
LIN {X -6.099,Y 99.757,Z 98,A 88.103,B 24.9184,C -2.0862,E1 24.9917,E2 -2.7212} C_DIS
LIN {X -3.5716,Y 99.8794,Z 98,A 86.5405,B 24.9187,C -2.0827,E1 24.9961,E2 -1.1499} C_DIS
LIN {X 1.7476,Y 99.9267,Z 98,A 83.9697,B 24.9172,C -2.1006,E1 25.0032,E2 1.3781} C_DIS
LIN {X 4.2579,Y 99.8512,Z 98,A 81.7357,B 24.9195,C -2.0719,E1 25.0096,E2 3.6796} C_DIS
LIN {X 7.5083,Y 99.6605,Z 98,A 80.1977,B 24.9186,C -2.0838,E1 25.0138,E2 5.1888} C_DIS
LIN {X 13.5449,Y 99.0211,Z 98,A 76.2061,B 24.9201,C -2.0645,E1 25.025,E2 9.223} C_DIS
LIN {X 17.3493,Y 98.4251,Z 98,A 74.8433,B 24.9177,C -2.0947,E1 25.0285,E2 10.513} C_DIS
LIN {X 19.8611,Y 97.9489,Z 98,A 73.0649,B 24.9187,C -2.0825,E1 25.0335,E2 12.318} C_DIS
LIN {X 23.0727,Y 97.244,Z 98,A 71.1168,B 24.9189,C -2.0792,E1 25.0388,E2 14.2714} C_DIS
LIN {X 26.8561,Y 96.2668,Z 98,A 68.9139,B 24.9189,C -2.0792,E1 25.0447,E2 16.4709} C_DIS
LIN {X 29.9712,Y 95.3429,Z 98,A 67.1706,B 24.9187,C -2.0822,E1 25.0493,E2 18.2039} C_DIS
LIN {X 32.084,Y 94.6522,Z 98,A 65.7893,B 24.9191,C -2.0771,E1 25.053,E2 19.5945} C_DIS
LIN {X 35.5562,Y 93.4033,Z 98,A 63.7625,B 24.919,C -2.0785,E1 25.0583,E2 21.6138} C_DIS
LIN {X 38.8742,Y 92.0716,Z 98,A 61.6961,B 24.9192,C -2.0757,E1 25.0636,E2 23.6821} C_DIS
LIN {X 42.6739,Y 90.3749,Z 98,A 59.4832,B 24.9189,C -2.0794,E1 25.0692,E2 25.8806} C_DIS
LIN {X 46.0859,Y 88.6835,Z 98,A 57.2965,B 24.9191,C -2.0765,E1 25.0747,E2 28.0682} C_DIS
LIN {X 48.7105,Y 87.2678,Z 98,A 55.4583,B 24.9197,C -2.0693,E1 25.0792,E2 29.9181} C_DIS
LIN {X 51.8756,Y 85.4243,Z 98,A 53.3539,B 24.92,C -2.0661,E1 25.0843,E2 32.0237} C_DIS
LIN {X 54.2681,Y 83.9254,Z 98,A 51.6662,B 24.9204,C -2.0609,E1 25.0883,E2 33.7182} C_DIS
LIN {X 57.0348,Y 82.0696,Z 98,A 49.992,B 24.9199,C -2.0668,E1 25.0921,E2 35.3729} C_DIS
LIN {X 59.27,Y 80.4707,Z 98,A 48.3345,B 24.9204,C -2.0609,E1 25.0959,E2 37.0384} C_DIS
LIN {X 61.2918,Y 78.942,Z 98,A 46.7417,B 24.921,C -2.0529,E1 25.0994,E2 38.6442} C_DIS
LIN {X 64.2063,Y 76.5906,Z 98,A 44.8254,B 24.9206,C -2.0577,E1 25.1035,E2 40.5419} C_DIS
LIN {X 66.1405,Y 74.9273,Z 98,A 43.0129,B 24.9219,C -2.0414,E1 25.1074,E2 42.3859} C_DIS
LIN {X 69.0735,Y 72.2315,Z 98,A 40.9765,B 24.9215,C -2.0462,E1 25.1115,E2 44.4024} C_DIS
LIN {X 71.3012,Y 70.0329,Z 98,A 39.3171,B 24.9214,C -2.0476,E1 25.1147,E2 46.0515} C_DIS
LIN {X 72.7525,Y 68.5235,Z 98,A 38.0123,B 24.9219,C -2.0409,E1 25.1173,E2 47.3664} C_DIS
LIN {X 74.4468,Y 66.6788,Z 98,A 36.5572,B 24.9222,C -2.037,E1 25.12,E2 48.8245} C_DIS
LIN {X 76.2959,Y 64.5557,Z 98,A 34.8636,B 24.9227,C -2.0301,E1 25.1231,E2 50.5265} C_DIS
LIN {X 78.4303,Y 61.9441,Z 98,A 33.0849,B 24.9227,C -2.0316,E1 25.1262,E2 52.2935} C_DIS
LIN {X 80.0271,Y 59.8673,Z 98,A 31.6793,B 24.9227,C -2.0316,E1 25.1286,E2 53.6923} C_DIS
LIN {X 81.6781,Y 57.5967,Z 98,A 29.8612,B 24.9235,C -2.0194,E1 25.1315,E2 55.5304} C_DIS
LIN {X 83.71,Y 54.601,Z 98,A 27.7827,B 24.9239,C -2.014,E1 25.1348,E2 57.6114} C_DIS
LIN {X 85.6761,Y 51.4613,Z 98,A 25.6707,B 24.9243,C -2.0089,E1 25.1378,E2 59.7249} C_DIS
LIN {X 87.5315,Y 48.2382,Z 98,A 23.7522,B 24.9241,C -2.0115,E1 25.1405,E2 61.6271} C_DIS
LIN {X 88.8304,Y 45.8004,Z 98,A 22.3038,B 24.9241,C -2.0125,E1 25.1423,E2 63.0655} C_DIS
LIN {X 90.3278,Y 42.7738,Z 98,A 20.0314,B 24.9255,C -1.9937,E1 25.1451,E2 65.37} C_DIS
LIN {X 91.8664,Y 39.3596,Z 98,A 17.933,B 24.9258,C -1.9895,E1 25.1475,E2 67.4669} C_DIS
LIN {X 93.2074,Y 36.0696,Z 98,A 15.9099,B 24.9262,C -1.9841,E1 25.1496,E2 69.4916} C_DIS
LIN {X 94.4417,Y 32.7006,Z 98,A 13.9719,B 24.9262,C -1.9828,E1 25.1514,E2 71.4219} C_DIS
LIN {X 95.4535,Y 29.6144,Z 98,A 12.0332,B 24.9269,C -1.9741,E1 25.1531,E2 73.37} C_DIS
LIN {X 96.3595,Y 26.5227,Z 98,A 10.291,B 24.927,C -1.9727,E1 25.1544,E2 75.1056} C_DIS
LIN {X 97.1396,Y 23.5016,Z 98,A 8.5716,B 24.9272,C -1.9699,E1 25.1555,E2 76.8216} C_DIS
LIN {X 97.6783,Y 21.151,Z 98,A 7.1442,B 24.9277,C -1.9639,E1 25.1564,E2 78.255} C_DIS
LIN {X 98.7383,Y 15.4649,Z 98,A 3.6254,B 24.929,C -1.9454,E1 25.1581,E2 81.7968} C_DIS
LIN {X 99.4041,Y 10.3542,Z 98,A 1.0746,B 24.9286,C -1.9522,E1 25.159,E2 84.3165} C_DIS
LIN {X 99.8453,Y 4.3945,Z 98,A -2.5469,B 24.9299,C -1.9333,E1 25.1597,E2 87.9609} C_DIS
LIN {X 99.9419,Y -0.2159,Z 98,A -4.891,B 24.9297,C -1.9368,E1 25.1597,E2 90.2828} C_DIS
LIN {X 99.865,Y -3.9371,Z 98,A -7.2861,B 24.9309,C -1.9195,E1 25.1597,E2 92.7047} C_DIS
LIN {X 99.6839,Y -7.1911,Z 98,A -9.2618,B 24.9317,C -1.9091,E1 25.1592,E2 94.693} C_DIS
LIN {X 99.2433,Y -11.7976,Z 98,A -11.6091,B 24.9314,C -1.9128,E1 25.1586,E2 97.0177} C_DIS
LIN {X 98.11,Y -19.0485,Z 98,A -15.6229,B 24.9318,C -1.907,E1 25.1568,E2 101.0215} C_DIS
LIN {X 97.0269,Y -23.9635,Z 98,A -18.7906,B 24.9333,C -1.8864,E1 25.1549,E2 104.2194} C_DIS
LIN {X 95.9999,Y -27.798,Z 98,A -20.961,B 24.9335,C -1.8834,E1 25.1533,E2 106.3844} C_DIS
LIN {X 95.3408,Y -29.9778,Z 98,A -22.4877,B 24.9344,C -1.8705,E1 25.152,E2 107.9331} C_DIS
LIN {X 94.3737,Y -32.8944,Z 98,A -24.0819,B 24.9344,C -1.8717,E1 25.1505,E2 109.5154} C_DIS
LIN {X 93.3371,Y -35.731,Z 98,A -25.7035,B 24.9344,C -1.8707,E1 25.149,E2 111.1302} C_DIS
LIN {X 92.1989,Y -38.5722,Z 98,A -27.397,B 24.9346,C -1.8678,E1 25.1472,E2 112.8212} C_DIS
LIN {X 91.3709,Y -40.4979,Z 98,A -28.6539,B 24.935,C -1.8619,E1 25.1458,E2 114.0852} C_DIS
LIN {X 90.2153,Y -43.0079,Z 98,A -30.7007,B 24.9366,C -1.8387,E1 25.1433,E2 116.1757} C_DIS
LIN {X 87.778,Y -47.7853,Z 98,A -33.267,B 24.9359,C -1.8499,E1 25.14,E2 118.7021} C_DIS
LIN {X 85.4164,Y -51.8886,Z 98,A -36.0626,B 24.9366,C -1.8387,E1 25.1361,E2 121.5096} C_DIS
LIN {X 83.5455,Y -54.8505,Z 98,A -38.0999,B 24.9371,C -1.8319,E1 25.133,E2 123.5527} C_DIS
LIN {X 81.5339,Y -57.7989,Z 98,A -40.1334,B 24.9375,C -1.8267,E1 25.1297,E2 125.5885} C_DIS
LIN {X 79.9824,Y -59.9267,Z 98,A -41.6946,B 24.9379,C -1.8206,E1 25.1271,E2 127.1567} C_DIS
LIN {X 78.1144,Y -62.3438,Z 98,A -43.2507,B 24.9377,C -1.8236,E1 25.1245,E2 128.6984} C_DIS
LIN {X 76.1506,Y -64.7262,Z 98,A -44.9642,B 24.9378,C -1.8212,E1 25.1214,E2 130.4096} C_DIS
LIN {X 74.1464,Y -67.0144,Z 98,A -46.884,B 24.9386,C -1.8098,E1 25.1178,E2 132.3479} C_DIS
LIN {X 72.1557,Y -69.1521,Z 98,A -48.3586,B 24.9384,C -1.8135,E1 25.115,E2 133.8072} C_DIS
LIN {X 70.6651,Y -70.6767,Z 98,A -49.6337,B 24.9387,C -1.8084,E1 25.1125,E2 135.089} C_DIS
LIN {X 69.1793,Y -72.1295,Z 98,A -50.7977,B 24.9388,C -1.8066,E1 25.1102,E2 136.2522} C_DIS
LIN {X 67.6189,Y -73.594,Z 98,A -52.168,B 24.9394,C -1.7981,E1 25.1073,E2 137.6372} C_DIS
LIN {X 64.9409,Y -75.9677,Z 98,A -54.1069,B 24.9394,C -1.7978,E1 25.1033,E2 139.5691} C_DIS
LIN {X 63.1532,Y -77.4606,Z 98,A -55.325,B 24.9394,C -1.7995,E1 25.1007,E2 140.7786} C_DIS
LIN {X 61.5409,Y -78.749,Z 98,A -56.5851,B 24.9397,C -1.7938,E1 25.0979,E2 142.0474} C_DIS
LIN {X 59.8785,Y -80.0187,Z 98,A -57.9917,B 24.9404,C -1.7832,E1 25.0947,E2 143.474} C_DIS
LIN {X 56.6365,Y -82.3464,Z 98,A -60.0691,B 24.9402,C -1.7867,E1 25.09,E2 145.5358} C_DIS
LIN {X 53.9826,Y -84.1086,Z 98,A -61.9863,B 24.9406,C -1.7796,E1 25.0855,E2 147.4635} C_DIS
LIN {X 50.8454,Y -86.0415,Z 98,A -64.0969,B 24.9409,C -1.7758,E1 25.0805,E2 149.5767} C_DIS
LIN {X 47.5819,Y -87.8883,Z 98,A -66.3028,B 24.9413,C -1.7698,E1 25.075,E2 151.7902} C_DIS
LIN {X 44.219,Y -89.6275,Z 98,A -68.2345,B 24.9409,C -1.7754,E1 25.0703,E2 153.7033} C_DIS
LIN {X 42.0399,Y -90.67,Z 98,A -70.2323,B 24.9426,C -1.7497,E1 25.0651,E2 155.757} C_DIS
LIN {X 38.963,Y -92.0342,Z 98,A -72.0998,B 24.9426,C -1.7492,E1 25.0603,E2 157.6211} C_DIS
LIN {X 35.9515,Y -93.2535,Z 98,A -73.4821,B 24.9416,C -1.7649,E1 25.0568,E2 158.9631} C_DIS
LIN {X 32.8231,Y -94.3987,Z 98,A -75.3231,B 24.9416,C -1.7651,E1 25.052,E2 160.8} C_DIS
LIN {X 30.8091,Y -95.0746,Z 98,A -76.7563,B 24.9422,C -1.7554,E1 25.0481,E2 162.2535} C_DIS
LIN {X 27.8526,Y -95.9842,Z 98,A -78.3373,B 24.9419,C -1.7607,E1 25.0439,E2 163.8192} C_DIS
LIN {X 25.7644,Y -96.5644,Z 98,A -79.6722,B 24.9422,C -1.7558,E1 25.0403,E2 165.1633} C_DIS
LIN {X 18.2861,Y -98.2567,Z 98,A -83.9623,B 24.9422,C -1.7558,E1 25.0286,E2 169.448} C_DIS
LIN {X 12.286,Y -99.1855,Z 98,A -87.5381,B 24.9426,C -1.7497,E1 25.0187,E2 173.0349} C_DIS
LIN {X 8.9651,Y -99.5393,Z 98,A -89.5138,B 24.9428,C -1.7464,E1 25.0132,E2 175.0172} C_DIS
LIN {X 4.2037,Y -99.8535,Z 98,A -92.3163,B 24.9431,C -1.7428,E1 25.0054,E2 177.8271} C_DIS
LIN {X 0.6838,Y -99.9382,Z 98,A -93.4768,B 24.941,C -1.7743,E1 25.0024,E2 178.9128} C_DIS
Enddeposition()
LIN {X 0.6838,Y -99.9382,Z 98,A -93.4768,B 24.941,C -1.7743,E1 25.0024,E2 178.9128} C_DIS
Startdeposition()
$VEL.CP = VEL_PRINT
LIN {X 1.728,Y -99.0314,Z 98,A -92.0858,B 24.9379,C -1.8196,E1 25.0065,E2 177.4146} C_DIS
LIN {X 6.0248,Y -98.8646,Z 98,A -90.4184,B 24.94,C -1.7896,E1 25.011,E2 175.8189} C_DIS
LIN {X 8.4707,Y -98.6838,Z 98,A -88.3584,B 24.9383,C -1.8146,E1 25.0169,E2 173.7008} C_DIS
LIN {X 12.0999,Y -98.3063,Z 98,A -86.8859,B 24.9398,C -1.7916,E1 25.0208,E2 172.2838} C_DIS
LIN {X 17.3836,Y -97.5091,Z 98,A -83.7748,B 24.9396,C -1.7946,E1 25.0294,E2 169.1686} C_DIS
LIN {X 23.5405,Y -96.2083,Z 98,A -80.0727,B 24.9393,C -1.8003,E1 25.0395,E2 165.4581} C_DIS
LIN {X 27.5375,Y -95.143,Z 98,A -77.743,B 24.9393,C -1.8003,E1 25.0458,E2 163.1319} C_DIS
LIN {X 30.4148,Y -94.261,Z 98,A -75.9269,B 24.9389,C -1.8054,E1 25.0506,E2 161.3073} C_DIS
LIN {X 33.6561,Y -93.1534,Z 98,A -74.2172,B 24.9394,C -1.7975,E1 25.0551,E2 159.6197} C_DIS
LIN {X 36.7825,Y -91.9649,Z 98,A -71.422,B 24.937,C -1.8334,E1 25.0626,E2 156.7456} C_DIS
LIN {X 40.2969,Y -90.479,Z 98,A -69.4733,B 24.9375,C -1.8267,E1 25.0675,E2 154.8176} C_DIS
LIN {X 43.7985,Y -88.8365,Z 98,A -67.1923,B 24.9371,C -1.832,E1 25.0732,E2 152.5301} C_DIS
LIN {X 46.646,Y -87.3765,Z 98,A -65.6851,B 24.9378,C -1.8217,E1 25.0769,E2 151.0515} C_DIS
LIN {X 49.3065,Y -85.9015,Z 98,A -64.0846,B 24.938,C -1.8187,E1 25.0807,E2 149.463} C_DIS
LIN {X 51.9614,Y -84.3242,Z 98,A -62.1087,B 24.9373,C -1.8294,E1 25.0855,E2 147.4679} C_DIS
LIN {X 56.2511,Y -81.5238,Z 98,A -59.2113,B 24.937,C -1.8327,E1 25.0922,E2 144.5723} C_DIS
LIN {X 59.0618,Y -79.5119,Z 98,A -57.2215,B 24.9368,C -1.8364,E1 25.0967,E2 142.5807} C_DIS
LIN {X 61.6902,Y -77.4896,Z 98,A -55.3597,B 24.9366,C -1.8384,E1 25.1008,E2 140.7212} C_DIS
LIN {X 64.2657,Y -75.3666,Z 98,A -53.4299,B 24.9364,C -1.8427,E1 25.1049,E2 138.7887} C_DIS
LIN {X 66.8849,Y -73.0521,Z 98,A -51.4209,B 24.9361,C -1.8469,E1 25.1091,E2 136.7779} C_DIS
LIN {X 69.4253,Y -70.6427,Z 98,A -49.7072,B 24.9366,C -1.8394,E1 25.1125,E2 135.0889} C_DIS
LIN {X 71.2568,Y -68.7944,Z 98,A -47.9129,B 24.9355,C -1.8545,E1 25.1161,E2 133.2666} C_DIS
LIN {X 73.5758,Y -66.3092,Z 98,A -45.8915,B 24.935,C -1.8617,E1 25.1199,E2 131.2372} C_DIS
LIN {X 75.9236,Y -63.6078,Z 98,A -43.8695,B 24.9348,C -1.8652,E1 25.1236,E2 129.2162} C_DIS
LIN {X 77.9856,Y -61.0627,Z 98,A -42.0081,B 24.9345,C -1.8689,E1 25.1268,E2 127.3547} C_DIS
LIN {X 80.1982,Y -58.1262,Z 98,A -39.4466,B 24.9329,C -1.8921,E1 25.1311,E2 124.7507} C_DIS
LIN {X 82.0823,Y -55.4321,Z 98,A -37.9883,B 24.9338,C -1.8796,E1 25.1333,E2 123.3291} C_DIS
LIN {X 83.9903,Y -52.496,Z 98,A -36.1466,B 24.9338,C -1.878,E1 25.1361,E2 121.5005} C_DIS
LIN {X 85.6609,Y -49.7253,Z 98,A -33.8891,B 24.9324,C -1.8989,E1 25.1393,E2 119.2053} C_DIS
LIN {X 89.2062,Y -43.0403,Z 98,A -29.7943,B 24.9323,C -1.9004,E1 25.1446,E2 115.1285} C_DIS
LIN {X 90.7294,Y -39.7291,Z 98,A -27.6939,B 24.9319,C -1.9065,E1 25.147,E2 113.0252} C_DIS
LIN {X 92.0024,Y -36.6881,Z 98,A -25.7656,B 24.9314,C -1.9132,E1 25.149,E2 111.0918} C_DIS
LIN {X 93.1184,Y -33.752,Z 98,A -24.0415,B 24.9312,C -1.9151,E1 25.1507,E2 109.3728} C_DIS
LIN {X 94.4205,Y -29.9221,Z 98,A -21.5979,B 24.9304,C -1.9266,E1 25.1528,E2 106.916} C_DIS
LIN {X 95.6431,Y -25.7412,Z 98,A -19.2025,B 24.9302,C -1.9295,E1 25.1546,E2 104.5273} C_DIS
LIN {X 96.2365,Y -23.4251,Z 98,A -17.5272,B 24.929,C -1.9457,E1 25.1558,E2 102.8235} C_DIS
LIN {X 97.1809,Y -19.1374,Z 98,A -14.2991,B 24.9264,C -1.9819,E1 25.1576,E2 99.5289} C_DIS
LIN {X 98.061,Y -13.9371,Z 98,A -12.2417,B 24.9286,C -1.9513,E1 25.1584,E2 97.5559} C_DIS
LIN {X 98.3707,Y -11.5503,Z 98,A -10.2221,B 24.9264,C -1.9812,E1 25.1591,E2 95.4776} C_DIS
LIN {X 98.7631,Y -7.4966,Z 98,A -8.6868,B 24.9283,C -1.9555,E1 25.1594,E2 94.012} C_DIS
LIN {X 98.9357,Y -4.7046,Z 98,A -6.8469,B 24.9273,C -1.9697,E1 25.1597,E2 92.1496} C_DIS
LIN {X 99.0357,Y -1.494,Z 98,A -4.1528,B 24.9243,C -2.0097,E1 25.1597,E2 89.3772} C_DIS
LIN {X 98.9814,Y 3.637,Z 98,A -2.2667,B 24.9268,C -1.9752,E1 25.1597,E2 87.5835} C_DIS
LIN {X 98.6189,Y 9.1933,Z 98,A 1.061,B 24.9258,C -1.9898,E1 25.159,E2 84.2412} C_DIS
LIN {X 98.1897,Y 13.0023,Z 98,A 3.7422,B 24.9238,C -2.0155,E1 25.158,E2 81.5152} C_DIS
LIN {X 97.6951,Y 16.3052,Z 98,A 5.5215,B 24.9238,C -2.0155,E1 25.1572,E2 79.7465} C_DIS
LIN {X 96.8134,Y 20.9142,Z 98,A 7.9587,B 24.924,C -2.0127,E1 25.1559,E2 77.33} C_DIS
LIN {X 95.9215,Y 24.6831,Z 98,A 10.0719,B 24.924,C -2.0145,E1 25.1545,E2 75.2248} C_DIS
LIN {X 95.0104,Y 27.9868,Z 98,A 12.059,B 24.9234,C -2.0207,E1 25.1529,E2 73.2344} C_DIS
LIN {X 94.1144,Y 30.8679,Z 98,A 14.2184,B 24.9218,C -2.0425,E1 25.1511,E2 71.0357} C_DIS
LIN {X 92.5362,Y 35.3173,Z 98,A 16.4969,B 24.9225,C -2.0325,E1 25.1489,E2 68.7938} C_DIS
LIN {X 91.312,Y 38.3708,Z 98,A 18.4512,B 24.922,C -2.04,E1 25.1468,E2 66.8324} C_DIS
LIN {X 90.3696,Y 40.5408,Z 98,A 20.4032,B 24.9199,C -2.0673,E1 25.1445,E2 64.8267} C_DIS
LIN {X 88.6895,Y 44.0952,Z 98,A 22.0663,B 24.9213,C -2.0492,E1 25.1425,E2 63.2151} C_DIS
LIN {X 86.4203,Y 48.3915,Z 98,A 24.9029,B 24.9206,C -2.0579,E1 25.1388,E2 60.3729} C_DIS
LIN {X 84.5383,Y 51.6092,Z 98,A 27.0265,B 24.9202,C -2.0623,E1 25.1357,E2 58.2497} C_DIS
LIN {X 82.8816,Y 54.2306,Z 98,A 29.2638,B 24.9185,C -2.0845,E1 25.1322,E2 55.9711} C_DIS
LIN {X 80.9116,Y 57.1293,Z 98,A 30.8552,B 24.9195,C -2.0724,E1 25.1297,E2 54.4163} C_DIS
LIN {X 79.0402,Y 59.6901,Z 98,A 32.8085,B 24.9187,C -2.0816,E1 25.1265,E2 52.4506} C_DIS
LIN {X 76.7414,Y 62.6184,Z 98,A 34.6648,B 24.9193,C -2.075,E1 25.1233,E2 50.6184} C_DIS
LIN {X 74.9979,Y 64.6984,Z 98,A 36.4146,B 24.9184,C -2.0857,E1 25.1201,E2 48.8514} C_DIS
LIN {X 71.6443,Y 68.3923,Z 98,A 39.2522,B 24.9181,C -2.0902,E1 25.1147,E2 46.0155} C_DIS
LIN {X 69.2476,Y 70.8182,Z 98,A 41.3007,B 24.9175,C -2.0973,E1 25.1106,E2 43.9589} C_DIS
LIN {X 64.9104,Y 74.8127,Z 98,A 44.5899,B 24.9173,C -2.0994,E1 25.1038,E2 40.6779} C_DIS
LIN {X 62.0881,Y 77.1711,Z 98,A 46.5784,B 24.9174,C -2.0981,E1 25.0995,E2 38.7002} C_DIS
LIN {X 58.4701,Y 79.9465,Z 98,A 49.2955,B 24.9168,C -2.1058,E1 25.0935,E2 35.9746} C_DIS
LIN {X 55.9784,Y 81.7123,Z 98,A 51.4171,B 24.9155,C -2.1224,E1 25.0885,E2 33.821} C_DIS
LIN {X 52.4675,Y 84.0081,Z 98,A 53.4849,B 24.9163,C -2.1124,E1 25.0837,E2 31.7835} C_DIS
LIN {X 49.3431,Y 85.8805,Z 98,A 55.4672,B 24.9164,C -2.1107,E1 25.079,E2 29.8112} C_DIS
LIN {X 47.1008,Y 87.1305,Z 98,A 57.3871,B 24.915,C -2.1293,E1 25.0742,E2 27.8528} C_DIS
LIN {X 42.8619,Y 89.292,Z 98,A 59.7647,B 24.9158,C -2.1185,E1 25.0683,E2 25.5073} C_DIS
LIN {X 38.9654,Y 91.0614,Z 98,A 62.3598,B 24.9152,C -2.1258,E1 25.0616,E2 22.9012} C_DIS
LIN {X 35.8179,Y 92.3442,Z 98,A 64.364,B 24.915,C -2.1292,E1 25.0564,E2 20.8935} C_DIS
LIN {X 32.5057,Y 93.5611,Z 98,A 66.6836,B 24.914,C -2.1415,E1 25.0503,E2 18.5494} C_DIS
LIN {X 27.9582,Y 95.0188,Z 98,A 69.0662,B 24.915,C -2.1293,E1 25.044,E2 16.2} C_DIS
LIN {X 24.6056,Y 95.9415,Z 98,A 71.0736,B 24.9149,C -2.1304,E1 25.0386,E2 14.1931} C_DIS
LIN {X 20.9307,Y 96.8098,Z 98,A 73.2893,B 24.9147,C -2.1327,E1 25.0325,E2 11.9749} C_DIS
LIN {X 17.3584,Y 97.5136,Z 98,A 75.2055,B 24.9152,C -2.1266,E1 25.0273,E2 10.0756} C_DIS
LIN {X 13.8919,Y 98.0674,Z 98,A 77.6326,B 24.914,C -2.1418,E1 25.0205,E2 7.6146} C_DIS
LIN {X 8.336,Y 98.696,Z 98,A 80.616,B 24.9147,C -2.1329,E1 25.0123,E2 4.6542} C_DIS
LIN {X 1.6746,Y 99.0324,Z 98,A 85.6367,B 24.9112,C -2.1754,E1 24.998,E2 -0.4662} C_DIS
LIN {X -4.4038,Y 98.9486,Z 98,A 87.6853,B 24.9157,C -2.1206,E1 24.9927,E2 -2.3852} C_DIS
LIN {X -9.2962,Y 98.6094,Z 98,A 90.8645,B 24.9148,C -2.1317,E1 24.9837,E2 -5.5919} C_DIS
LIN {X -14.5821,Y 97.9687,Z 98,A 93.9823,B 24.9148,C -2.1311,E1 24.9751,E2 -8.7107} C_DIS
LIN {X -18.0295,Y 97.393,Z 98,A 95.9931,B 24.915,C -2.1292,E1 24.9696,E2 -10.7189} C_DIS
LIN {X -21.499,Y 96.6858,Z 98,A 98.0125,B 24.9152,C -2.1264,E1 24.9641,E2 -12.7341} C_DIS
LIN {X -24.862,Y 95.8756,Z 98,A 99.7761,B 24.916,C -2.1161,E1 24.9593,E2 -14.4756} C_DIS
LIN {X -27.796,Y 95.067,Z 98,A 101.5171,B 24.9162,C -2.1135,E1 24.9547,E2 -16.2133} C_DIS
LIN {X -31.9314,Y 93.7586,Z 98,A 104.3596,B 24.9155,C -2.1223,E1 24.9471,E2 -19.0819} C_DIS
LIN {X -35.4696,Y 92.4785,Z 98,A 106.4964,B 24.9159,C -2.118,E1 24.9415,E2 -21.2129} C_DIS
LIN {X -38.7619,Y 91.1472,Z 98,A 108.2438,B 24.9169,C -2.1044,E1 24.937,E2 -22.9319} C_DIS
LIN {X -43.3615,Y 89.0519,Z 98,A 111.5303,B 24.9163,C -2.1125,E1 24.9287,E2 -26.2459} C_DIS
LIN {X -46.1799,Y 87.622,Z 98,A 113.4831,B 24.9162,C -2.1139,E1 24.9238,E2 -28.2073} C_DIS
LIN {X -51.4605,Y 84.6287,Z 98,A 116.9253,B 24.9169,C -2.1052,E1 24.9155,E2 -31.639} C_DIS
LIN {X -54.4407,Y 82.7431,Z 98,A 119.1951,B 24.9166,C -2.1092,E1 24.9102,E2 -33.9258} C_DIS
LIN {X -58.4771,Y 79.9414,Z 98,A 121.8202,B 24.9176,C -2.0959,E1 24.9042,E2 -36.5284} C_DIS
LIN {X -61.3484,Y 77.7597,Z 98,A 123.7984,B 24.9183,C -2.0878,E1 24.8999,E2 -38.4945} C_DIS
LIN {X -63.3561,Y 76.1329,Z 98,A 125.7808,B 24.9172,C -2.1013,E1 24.8956,E2 -40.5165} C_DIS
LIN {X -65.9559,Y 73.892,Z 98,A 127.519,B 24.9182,C -2.0882,E1 24.892,E2 -42.2305} C_DIS
LIN {X -69.0069,Y 71.052,Z 98,A 129.8032,B 24.919,C -2.0782,E1 24.8874,E2 -44.5002} C_DIS
LIN {X -71.6966,Y 68.3381,Z 98,A 132.4249,B 24.9183,C -2.0868,E1 24.8823,E2 -47.1538} C_DIS
LIN {X -73.9774,Y 65.8606,Z 98,A 134.0109,B 24.9197,C -2.0695,E1 24.8794,E2 -48.7058} C_DIS
LIN {X -77.2579,Y 61.9811,Z 98,A 136.9223,B 24.9204,C -2.0609,E1 24.8742,E2 -51.6101} C_DIS
LIN {X -80.28,Y 58.0118,Z 98,A 140.0263,B 24.9204,C -2.0605,E1 24.869,E2 -54.7281} C_DIS
LIN {X -84.3807,Y 51.8686,Z 98,A 144.107,B 24.9218,C -2.042,E1 24.8628,E2 -58.7852} C_DIS
LIN {X -86.0026,Y 49.1305,Z 98,A 145.9444,B 24.9222,C -2.0366,E1 24.8602,E2 -60.6192} C_DIS
LIN {X -87.7147,Y 46.0039,Z 98,A 147.9853,B 24.9227,C -2.0299,E1 24.8576,E2 -62.6548} C_DIS
LIN {X -89.277,Y 42.893,Z 98,A 150.104,B 24.9229,C -2.0274,E1 24.8549,E2 -64.7791} C_DIS
LIN {X -91.5257,Y 37.8616,Z 98,A 153.8191,B 24.9223,C -2.0354,E1 24.8508,E2 -68.534} C_DIS
LIN {X -92.9177,Y 34.3023,Z 98,A 156.513,B 24.9216,C -2.045,E1 24.8482,E2 -71.266} C_DIS
LIN {X -94.7054,Y 29.0034,Z 98,A 158.6708,B 24.9251,C -1.9986,E1 24.8465,E2 -73.3252} C_DIS
LIN {X -95.9534,Y 24.5592,Z 98,A 161.3576,B 24.9257,C -1.9907,E1 24.8445,E2 -76.0089} C_DIS
LIN {X -96.7536,Y 21.1884,Z 98,A 163.3512,B 24.9262,C -1.984,E1 24.8433,E2 -77.9982} C_DIS
LIN {X -97.3199,Y 18.4158,Z 98,A 165.6176,B 24.925,C -1.9998,E1 24.8421,E2 -80.3157} C_DIS
LIN {X -97.9412,Y 14.76,Z 98,A 167.294,B 24.9267,C -1.9772,E1 24.8414,E2 -81.9482} C_DIS
LIN {X -98.353,Y 11.701,Z 98,A 169.0523,B 24.9272,C -1.9705,E1 24.8407,E2 -83.7011} C_DIS
LIN {X -98.718,Y 8.0615,Z 98,A 171.174,B 24.9277,C -1.9639,E1 24.8402,E2 -85.8197} C_DIS
LIN {X -98.9429,Y 4.5375,Z 98,A 173.2086,B 24.9282,C -1.9571,E1 24.8399,E2 -87.8502} C_DIS
LIN {X -99.0377,Y 1.3868,Z 98,A 175.1072,B 24.9284,C -1.9537,E1 24.8398,E2 -89.7522} C_DIS
LIN {X -99.0405,Y -1.2364,Z 98,A 176.6623,B 24.9287,C -1.9501,E1 24.8398,E2 -91.308} C_DIS
LIN {X -98.9319,Y -4.7921,Z 98,A 178.8182,B 24.9289,C -1.9468,E1 24.8401,E2 -93.4691} C_DIS
LIN {X -98.6438,Y -8.9239,Z 98,A -178.9828,B 24.93,C -1.9326,E1 24.8406,E2 -95.6474} C_DIS
LIN {X -98.3011,Y -12.1426,Z 98,A -176.9606,B 24.93,C -1.9316,E1 24.8412,E2 -97.6794} C_DIS
LIN {X -97.7866,Y -15.7579,Z 98,A -174.5003,B 24.9297,C -1.9367,E1 24.8423,E2 -100.1664} C_DIS
LIN {X -96.9086,Y -20.4754,Z 98,A -172.0783,B 24.9312,C -1.9161,E1 24.8436,E2 -102.5537} C_DIS
LIN {X -96.174,Y -23.6813,Z 98,A -170.2497,B 24.9318,C -1.9078,E1 24.8448,E2 -104.3732} C_DIS
LIN {X -95.109,Y -27.6542,Z 98,A -167.9696,B 24.9325,C -1.8972,E1 24.8464,E2 -106.6412} C_DIS
LIN {X -93.7882,Y -31.8437,Z 98,A -165.1428,B 24.9324,C -1.8992,E1 24.8489,E2 -109.4891} C_DIS
LIN {X -92.4177,Y -35.6272,Z 98,A -162.7299,B 24.9327,C -1.8953,E1 24.8513,E2 -111.9061} C_DIS
LIN {X -90.8231,Y -39.5141,Z 98,A -160.4604,B 24.9335,C -1.8828,E1 24.8537,E2 -114.1585} C_DIS
LIN {X -89.5481,Y -42.3281,Z 98,A -158.5995,B 24.9337,C -1.8803,E1 24.8559,E2 -116.0234} C_DIS
LIN {X -86.2464,Y -48.7029,Z 98,A -154.5537,B 24.9348,C -1.8652,E1 24.8612,E2 -120.0548} C_DIS
LIN {X -83.8524,Y -52.7167,Z 98,A -151.7129,B 24.935,C -1.8628,E1 24.8653,E2 -122.9044} C_DIS
LIN {X -82.114,Y -55.3852,Z 98,A -149.9259,B 24.9354,C -1.8562,E1 24.8681,E2 -124.6846} C_DIS
LIN {X -77.6094,Y -61.5386,Z 98,A -145.5115,B 24.9362,C -1.8454,E1 24.8754,E2 -129.0946} C_DIS
LIN {X -73.6115,Y -66.2693,Z 98,A -141.9337,B 24.9367,C -1.8369,E1 24.8819,E2 -132.6685} C_DIS
LIN {X -71.4925,Y -68.5499,Z 98,A -140.0178,B 24.9367,C -1.837,E1 24.8856,E2 -134.5929} C_DIS
LIN {X -66.813,Y -73.1181,Z 98,A -136.1944,B 24.9372,C -1.8306,E1 24.8933,E2 -138.4168} C_DIS
LIN {X -64.4668,Y -75.1952,Z 98,A -133.7523,B 24.9359,C -1.8492,E1 24.8986,E2 -140.9129} C_DIS
LIN {X -61.1674,Y -77.9028,Z 98,A -131.8981,B 24.9377,C -1.823,E1 24.9026,E2 -142.7115} C_DIS
LIN {X -58.3758,Y -80.0156,Z 98,A -129.3047,B 24.9366,C -1.8396,E1 24.9085,E2 -145.3536} C_DIS
LIN {X -55.0124,Y -82.3661,Z 98,A -127.5655,B 24.9384,C -1.8132,E1 24.9124,E2 -147.0358} C_DIS
LIN {X -52.3351,Y -84.0908,Z 98,A -125.7095,B 24.9385,C -1.8109,E1 24.9168,E2 -148.8922} C_DIS
LIN {X -47.8141,Y -86.7428,Z 98,A -122.5774,B 24.9385,C -1.8102,E1 24.9244,E2 -152.0319} C_DIS
LIN {X -44.7578,Y -88.3576,Z 98,A -120.8995,B 24.9395,C -1.7962,E1 24.9285,E2 -153.681} C_DIS
LIN {X -41.8019,Y -89.7931,Z 98,A -118.7609,B 24.9391,C -1.8024,E1 24.9339,E2 -155.8399} C_DIS
LIN {X -38.3858,Y -91.3057,Z 98,A -116.5682,B 24.9391,C -1.8013,E1 24.9395,E2 -158.035} C_DIS
LIN {X -35.8153,Y -92.3452,Z 98,A -114.5773,B 24.9383,C -1.8137,E1 24.9448,E2 -160.0597} C_DIS
LIN {X -31.329,Y -93.9617,Z 98,A -112.21,B 24.9395,C -1.7972,E1 24.951,E2 -162.3923} C_DIS
LIN {X -28.6648,Y -94.8092,Z 98,A -109.9482,B 24.9379,C -1.8196,E1 24.9572,E2 -164.7112} C_DIS
LIN {X -24.7862,Y -95.895,Z 98,A -107.9781,B 24.9389,C -1.805,E1 24.9624,E2 -166.6496} C_DIS
LIN {X -20.2374,Y -96.9575,Z 98,A -105.8249,B 24.9404,C -1.7836,E1 24.9681,E2 -168.7546} C_DIS
LIN {X -15.8839,Y -97.7656,Z 98,A -102.1914,B 24.9378,C -1.8224,E1 24.9784,E2 -172.4838} C_DIS
LIN {X -11.2857,Y -98.4017,Z 98,A -100.4549,B 24.9402,C -1.7866,E1 24.983,E2 -174.1367} C_DIS
LIN {X -6.8081,Y -98.8123,Z 98,A -97.6823,B 24.9398,C -1.7929,E1 24.9907,E2 -176.9254} C_DIS
LIN {X -0.8931,Y -99.0428,Z 98,A -94.3502,B 24.94,C -1.7899,E1 25,E2 -180.2508} C_DIS
LIN {X -0.8931,Y -99.0428,Z 98,A -94.3502,B 24.94,C -1.7899,E1 25,E2 -180.2508} C_DIS
Enddeposition()
LIN {X 0.6899,Y -98.1442,Z 98,A -95.1492,B 24.943,C -1.7432,E1 24.9975,E2 -179.3413} C_DIS
Startdeposition()
$VEL.CP = VEL_PRINT
LIN {X -4.3621,Y -98.0541,Z 98,A -96.7069,B 24.9397,C -1.7931,E1 24.9935,E2 -177.9015} C_DIS
LIN {X -9.1489,Y -97.7237,Z 98,A -99.7269,B 24.9403,C -1.785,E1 24.985,E2 -174.8612} C_DIS
LIN {X -11.6852,Y -97.4533,Z 98,A -102.0794,B 24.9423,C -1.7542,E1 24.9783,E2 -172.4341} C_DIS
LIN {X -15.4023,Y -96.9358,Z 98,A -104.0848,B 24.9419,C -1.7614,E1 24.9728,E2 -170.4439} C_DIS
LIN {X -19.544,Y -96.1856,Z 98,A -106.1708,B 24.9409,C -1.7755,E1 24.9671,E2 -168.3893} C_DIS
LIN {X -22.6522,Y -95.503,Z 98,A -108.6414,B 24.9423,C -1.7548,E1 24.9603,E2 -165.866} C_DIS
LIN {X -26.3881,Y -94.5378,Z 98,A -110.2433,B 24.9407,C -1.7791,E1 24.9561,E2 -164.3195} C_DIS
LIN {X -28.7542,Y -93.8452,Z 98,A -111.9719,B 24.9413,C -1.7699,E1 24.9514,E2 -162.5661} C_DIS
LIN {X -32.3587,Y -92.6636,Z 98,A -114.7634,B 24.9425,C -1.7517,E1 24.9439,E2 -159.7259} C_DIS
LIN {X -36.7497,Y -91.0118,Z 98,A -116.3942,B 24.9397,C -1.7929,E1 24.9399,E2 -158.1896} C_DIS
LIN {X -42.1815,Y -88.6254,Z 98,A -119.9139,B 24.9397,C -1.7947,E1 24.9309,E2 -154.6657} C_DIS
LIN {X -44.1811,Y -87.6467,Z 98,A -121.5386,B 24.9403,C -1.7849,E1 24.9268,E2 -153.0134} C_DIS
LIN {X -47.4096,Y -85.943,Z 98,A -124.6015,B 24.9422,C -1.7559,E1 24.9191,E2 -149.8726} C_DIS
LIN {X -51.9776,Y -83.2583,Z 98,A -127.2177,B 24.9408,C -1.7767,E1 24.913,E2 -147.2978} C_DIS
LIN {X -54.9512,Y -81.3264,Z 98,A -129.1607,B 24.9403,C -1.7844,E1 24.9085,E2 -145.3666} C_DIS
LIN {X -58.9774,Y -78.4556,Z 98,A -131.6567,B 24.9391,C -1.8026,E1 24.903,E2 -142.9053} C_DIS
LIN {X -64.4179,Y -74.054,Z 98,A -135.6904,B 24.9385,C -1.812,E1 24.8943,E2 -138.8786} C_DIS
LIN {X -69.9972,Y -68.8045,Z 98,A -140.1793,B 24.9379,C -1.8206,E1 24.8852,E2 -134.3916} C_DIS
LIN {X -72.2241,Y -66.4629,Z 98,A -142.8492,B 24.9394,C -1.7985,E1 24.88,E2 -131.6574} C_DIS
LIN {X -74.9852,Y -63.3321,Z 98,A -144.4738,B 24.9371,C -1.8312,E1 24.8772,E2 -130.1033} C_DIS
LIN {X -76.4861,Y -61.5112,Z 98,A -146.3135,B 24.938,C -1.819,E1 24.8739,E2 -128.2259} C_DIS
LIN {X -80.2586,Y -56.5023,Z 98,A -149.5569,B 24.9364,C -1.8419,E1 24.8686,E2 -125.0213} C_DIS
LIN {X -82.7637,Y -52.7625,Z 98,A -152.2759,B 24.9362,C -1.8456,E1 24.8644,E2 -122.2975} C_DIS
LIN {X -84.5065,Y -49.9225,Z 98,A -154.2252,B 24.9358,C -1.8506,E1 24.8616,E2 -120.3501} C_DIS
LIN {X -86.0987,Y -47.1241,Z 98,A -156.6223,B 24.9366,C -1.8386,E1 24.8583,E2 -117.9119} C_DIS
LIN {X -87.6727,Y -44.1302,Z 98,A -158.043,B 24.935,C -1.8622,E1 24.8566,E2 -116.5399} C_DIS
LIN {X -89.4538,Y -40.3936,Z 98,A -160.5675,B 24.9348,C -1.8655,E1 24.8535,E2 -114.0094} C_DIS
LIN {X -90.8285,Y -37.1999,Z 98,A -162.7121,B 24.9346,C -1.8676,E1 24.8512,E2 -111.8579} C_DIS
LIN {X -92.4408,Y -32.9938,Z 98,A -165.8197,B 24.9352,C -1.8597,E1 24.8482,E2 -108.714} C_DIS
LIN {X -93.5815,Y -29.6011,Z 98,A -167.3356,B 24.9334,C -1.8846,E1 24.8469,E2 -107.2489} C_DIS
LIN {X -95.1119,Y -24.2358,Z 98,A -170.5995,B 24.9327,C -1.8943,E1 24.8445,E2 -103.9891} C_DIS
LIN {X -95.7744,Y -21.4754,Z 98,A -172.448,B 24.9328,C -1.8931,E1 24.8433,E2 -102.127} C_DIS
LIN {X -96.9001,Y -15.6303,Z 98,A -175.655,B 24.9314,C -1.9127,E1 24.8417,E2 -98.9477} C_DIS
LIN {X -97.4111,Y -12.042,Z 98,A -177.9433,B 24.9314,C -1.9138,E1 24.8409,E2 -96.6482} C_DIS
LIN {X -97.7495,Y -8.8699,Z 98,A -179.7861,B 24.9309,C -1.9203,E1 24.8403,E2 -94.81} C_DIS
LIN {X -98.0362,Y -4.7772,Z 98,A 177.7743,B 24.9304,C -1.9265,E1 24.8399,E2 -92.3704} C_DIS
LIN {X -98.1307,Y -2.0043,Z 98,A 176.1518,B 24.93,C -1.9316,E1 24.8398,E2 -90.7504} C_DIS
LIN {X -98.1436,Y 1.3053,Z 98,A 174.0063,B 24.9301,C -1.9309,E1 24.8398,E2 -88.5903} C_DIS
LIN {X -97.9915,Y 5.5945,Z 98,A 171.638,B 24.9292,C -1.9434,E1 24.8401,E2 -86.2377} C_DIS
LIN {X -97.7468,Y 8.8985,Z 98,A 169.7405,B 24.9286,C -1.9508,E1 24.8406,E2 -84.3464} C_DIS
LIN {X -97.3698,Y 12.3613,Z 98,A 167.6156,B 24.9284,C -1.9544,E1 24.8412,E2 -82.2173} C_DIS
LIN {X -96.1631,Y 19.6541,Z 98,A 163.7059,B 24.9264,C -1.9814,E1 24.8431,E2 -78.3487} C_DIS
LIN {X -95.3274,Y 23.3734,Z 98,A 160.2239,B 24.9289,C -1.9479,E1 24.8454,E2 -74.7665} C_DIS
LIN {X -94.0858,Y 27.9547,Z 98,A 158.0519,B 24.9268,C -1.9758,E1 24.847,E2 -72.6484} C_DIS
LIN {X -92.3362,Y 33.2834,Z 98,A 155.2231,B 24.925,C -2.0004,E1 24.8495,E2 -69.8622} C_DIS
LIN {X -91.4001,Y 35.7723,Z 98,A 152.6237,B 24.9271,C -1.9714,E1 24.8522,E2 -67.179} C_DIS
LIN {X -89.6284,Y 40.0061,Z 98,A 150.3321,B 24.9256,C -1.9919,E1 24.8548,E2 -64.9237} C_DIS
LIN {X -87.7309,Y 44.0128,Z 98,A 148.1974,B 24.9239,C -2.0143,E1 24.8573,E2 -62.8309} C_DIS
LIN {X -86.0882,Y 47.1442,Z 98,A 146.0622,B 24.9236,C -2.018,E1 24.8601,E2 -60.6933} C_DIS
LIN {X -84.4786,Y 49.9698,Z 98,A 144.0801,B 24.9234,C -2.0208,E1 24.8629,E2 -58.7074} C_DIS
LIN {X -81.3478,Y 54.9196,Z 98,A 139.6654,B 24.9251,C -1.9981,E1 24.8698,E2 -54.2166} C_DIS
LIN {X -78.1761,Y 59.3494,Z 98,A 137.6361,B 24.9217,C -2.0441,E1 24.873,E2 -52.287} C_DIS
LIN {X -75.4498,Y 62.777,Z 98,A 134.7672,B 24.9219,C -2.0405,E1 24.8781,E2 -49.3963} C_DIS
LIN {X -70.5955,Y 68.1902,Z 98,A 130.6631,B 24.9207,C -2.0558,E1 24.8858,E2 -45.3104} C_DIS
LIN {X -66.5839,Y 72.113,Z 98,A 127.6322,B 24.9195,C -2.0717,E1 24.8918,E2 -42.3048} C_DIS
LIN {X -62.0993,Y 76.0094,Z 98,A 124.103,B 24.9191,C -2.0774,E1 24.8993,E2 -38.7753} C_DIS
LIN {X -57.8743,Y 79.2729,Z 98,A 120.2039,B 24.9206,C -2.0578,E1 24.9081,E2 -34.8157} C_DIS
LIN {X -54.9197,Y 81.3478,Z 98,A 119.0371,B 24.9178,C -2.0935,E1 24.9106,E2 -33.7298} C_DIS
LIN {X -52.9613,Y 82.6361,Z 98,A 117.2719,B 24.9187,C -2.0827,E1 24.9148,E2 -31.9332} C_DIS
LIN {X -47.9968,Y 85.6151,Z 98,A 113.918,B 24.9181,C -2.0896,E1 24.9229,E2 -28.5857} C_DIS
LIN {X -46.0637,Y 86.6711,Z 98,A 112.611,B 24.918,C -2.0911,E1 24.9261,E2 -27.2785} C_DIS
LIN {X -43.4715,Y 87.9992,Z 98,A 110.3594,B 24.9192,C -2.0752,E1 24.9318,E2 -24.9833} C_DIS
LIN {X -40.3332,Y 89.4809,Z 98,A 108.4011,B 24.9188,C -2.0806,E1 24.9368,E2 -23.0328} C_DIS
LIN {X -37.3539,Y 90.7659,Z 98,A 106.9298,B 24.9175,C -2.0976,E1 24.9405,E2 -21.5986} C_DIS
LIN {X -34.3217,Y 91.9557,Z 98,A 104.5418,B 24.9186,C -2.0835,E1 24.9468,E2 -19.1722} C_DIS
LIN {X -31.1726,Y 93.0694,Z 98,A 102.8264,B 24.9178,C -2.0939,E1 24.9513,E2 -17.4782} C_DIS
LIN {X -28.2348,Y 94.0027,Z 98,A 100.8265,B 24.9182,C -2.089,E1 24.9567,E2 -15.4633} C_DIS
LIN {X -25.0687,Y 94.8971,Z 98,A 99.3998,B 24.9167,C -2.1079,E1 24.9604,E2 -14.0794} C_DIS
LIN {X -22.456,Y 95.5483,Z 98,A 97.6481,B 24.917,C -2.1032,E1 24.9652,E2 -12.3141} C_DIS
LIN {X -19.0423,Y 96.2873,Z 98,A 95.7342,B 24.9166,C -2.1092,E1 24.9704,E2 -10.4123} C_DIS
LIN {X -16.4661,Y 96.7603,Z 98,A 94.1312,B 24.9166,C -2.1078,E1 24.9748,E2 -8.8044} C_DIS
LIN {X -12.8619,Y 97.3049,Z 98,A 91.776,B 24.9172,C -2.1013,E1 24.9814,E2 -6.4317} C_DIS
LIN {X -8.9977,Y 97.7377,Z 98,A 89.4679,B 24.9172,C -2.1011,E1 24.9878,E2 -4.1219} C_DIS
LIN {X -3.7311,Y 98.0812,Z 98,A 85.8569,B 24.9186,C -2.0837,E1 24.998,E2 -0.4688} C_DIS
LIN {X 1.0017,Y 98.1467,Z 98,A 84.1734,B 24.9155,C -2.1221,E1 25.0025,E2 1.1233} C_DIS
LIN {X 5.4441,Y 97.9999,Z 98,A 81.3727,B 24.9161,C -2.115,E1 25.0103,E2 3.9404} C_DIS
LIN {X 8.8965,Y 97.747,Z 98,A 78.5953,B 24.9182,C -2.088,E1 25.0182,E2 6.7802} C_DIS
LIN {X 13.238,Y 97.2555,Z 98,A 76.9138,B 24.9158,C -2.1184,E1 25.0227,E2 8.3883} C_DIS
LIN {X 15.7285,Y 96.8836,Z 98,A 75.2437,B 24.9164,C -2.1107,E1 25.0273,E2 10.075} C_DIS
LIN {X 18.9768,Y 96.2999,Z 98,A 73.288,B 24.9166,C -2.1089,E1 25.0327,E2 12.0327} C_DIS
LIN {X 22.5255,Y 95.5322,Z 98,A 71.2562,B 24.9164,C -2.111,E1 25.0382,E2 14.0568} C_DIS
LIN {X 25.523,Y 94.7744,Z 98,A 69.2335,B 24.9171,C -2.102,E1 25.0437,E2 16.0977} C_DIS
LIN {X 29.066,Y 93.7485,Z 98,A 66.4711,B 24.919,C -2.0784,E1 25.0512,E2 18.9111} C_DIS
LIN {X 33.5497,Y 92.239,Z 98,A 64.585,B 24.9167,C -2.1076,E1 25.056,E2 20.724} C_DIS
LIN {X 39.3044,Y 89.9377,Z 98,A 61.1108,B 24.9166,C -2.1092,E1 25.065,E2 24.1865} C_DIS
LIN {X 41.1655,Y 89.1016,Z 98,A 59.6857,B 24.9174,C -2.0992,E1 25.0686,E2 25.6319} C_DIS
LIN {X 44.4378,Y 87.5154,Z 98,A 56.9439,B 24.9194,C -2.0737,E1 25.0756,E2 28.4264} C_DIS
LIN {X 48.1454,Y 85.5321,Z 98,A 55.1587,B 24.9177,C -2.095,E1 25.0798,E2 30.156} C_DIS
LIN {X 51.1658,Y 83.7599,Z 98,A 52.3874,B 24.92,C -2.0651,E1 25.0866,E2 32.9896} C_DIS
LIN {X 54.9133,Y 81.3521,Z 98,A 50.5683,B 24.9181,C -2.0898,E1 25.0907,E2 34.7439} C_DIS
LIN {X 57.6702,Y 79.4224,Z 98,A 47.7329,B 24.9209,C -2.054,E1 25.0972,E2 37.654} C_DIS
LIN {X 61.5248,Y 76.4751,Z 98,A 45.9289,B 24.9183,C -2.0873,E1 25.101,E2 39.3728} C_DIS
LIN {X 63.6705,Y 74.6972,Z 98,A 43.2991,B 24.9215,C -2.0465,E1 25.1068,E2 42.0887} C_DIS
LIN {X 67.2688,Y 71.474,Z 98,A 41.7247,B 24.9183,C -2.0877,E1 25.1098,E2 43.5593} C_DIS
LIN {X 69.1482,Y 69.6577,Z 98,A 39.7388,B 24.9199,C -2.067,E1 25.1138,E2 45.586} C_DIS
LIN {X 73.7118,Y 64.8097,Z 98,A 35.9217,B 24.9203,C -2.0609,E1 25.1211,E2 49.4005} C_DIS
LIN {X 75.8478,Y 62.2979,Z 98,A 33.5276,B 24.9221,C -2.0385,E1 25.1254,E2 51.8364} C_DIS
LIN {X 78.052,Y 59.5126,Z 98,A 31.8978,B 24.9212,C -2.0504,E1 25.1281,E2 53.4305} C_DIS
LIN {X 80.1882,Y 56.6014,Z 98,A 28.9084,B 24.9241,C -2.0116,E1 25.1331,E2 56.497} C_DIS
LIN {X 83.102,Y 52.2278,Z 98,A 26.8589,B 24.9218,C -2.0425,E1 25.136,E2 58.4633} C_DIS
LIN {X 84.8099,Y 49.4088,Z 98,A 24.1728,B 24.9244,C -2.0081,E1 25.1399,E2 61.2168} C_DIS
LIN {X 86.9221,Y 45.5871,Z 98,A 22.3183,B 24.9229,C -2.0278,E1 25.1423,E2 63.015} C_DIS
LIN {X 88.6833,Y 42.06,Z 98,A 19.0824,B 24.9261,C -1.9854,E1 25.1463,E2 66.3336} C_DIS
LIN {X 90.868,Y 37.1029,Z 98,A 17.338,B 24.9226,C -2.031,E1 25.148,E2 67.9607} C_DIS
LIN {X 93.2919,Y 30.5011,Z 98,A 12.9269,B 24.9245,C -2.0069,E1 25.1523,E2 72.404} C_DIS
LIN {X 94.0701,Y 28.0077,Z 98,A 11.3954,B 24.9248,C -2.0021,E1 25.1535,E2 73.9382} C_DIS
LIN {X 94.9684,Y 24.7943,Z 98,A 9.3957,B 24.9254,C -1.9941,E1 25.155,E2 75.9452} C_DIS
LIN {X 95.79,Y 21.4039,Z 98,A 7.3244,B 24.926,C -1.9864,E1 25.1563,E2 78.0226} C_DIS
LIN {X 96.4881,Y 17.9995,Z 98,A 5.2324,B 24.9267,C -1.9776,E1 25.1574,E2 80.1232} C_DIS
LIN {X 97.4482,Y 11.7288,Z 98,A 1.714,B 24.927,C -1.9732,E1 25.1588,E2 83.6313} C_DIS
LIN {X 97.7888,Y 8.4428,Z 98,A -0.9673,B 24.9296,C -1.9376,E1 25.1595,E2 86.3805} C_DIS
LIN {X 98.0688,Y 4.0189,Z 98,A -2.2317,B 24.9264,C -1.9812,E1 25.1597,E2 87.5346} C_DIS
LIN {X 98.1319,Y -1.9386,Z 98,A -5.7264,B 24.9273,C -1.9693,E1 25.1597,E2 91.0366} C_DIS
LIN {X 97.88,Y -7.3063,Z 98,A -9.7915,B 24.9307,C -1.9226,E1 25.1591,E2 95.1879} C_DIS
LIN {X 97.5807,Y -10.5706,Z 98,A -11.0577,B 24.9293,C -1.9418,E1 25.1588,E2 96.4011} C_DIS
LIN {X 97.2694,Y -13.1356,Z 98,A -12.8319,B 24.9304,C -1.9265,E1 25.1581,E2 98.2011} C_DIS
LIN {X 96.2508,Y -19.2265,Z 98,A -16.6657,B 24.9319,C -1.9059,E1 25.1562,E2 102.0608} C_DIS
LIN {X 95.4461,Y -22.8867,Z 98,A -18.4944,B 24.9314,C -1.913,E1 25.1551,E2 103.8622} C_DIS
LIN {X 94.6375,Y -26.0301,Z 98,A -20.8016,B 24.933,C -1.8909,E1 25.1534,E2 106.2085} C_DIS
LIN {X 93.3759,Y -30.2416,Z 98,A -22.9234,B 24.9323,C -1.9002,E1 25.1517,E2 108.2961} C_DIS
LIN {X 92.2107,Y -33.6273,Z 98,A -24.9788,B 24.9327,C -1.8951,E1 25.1497,E2 110.352} C_DIS
LIN {X 90.9673,Y -36.8591,Z 98,A -27.0325,B 24.9332,C -1.8876,E1 25.1476,E2 112.412} C_DIS
LIN {X 89.5387,Y -40.2051,Z 98,A -28.9081,B 24.933,C -1.8909,E1 25.1456,E2 114.2696} C_DIS
LIN {X 88.4241,Y -42.6004,Z 98,A -30.7423,B 24.9341,C -1.8748,E1 25.1433,E2 116.1319} C_DIS
LIN {X 86.0484,Y -47.2176,Z 98,A -34.0451,B 24.9355,C -1.8552,E1 25.139,E2 119.4635} C_DIS
LIN {X 83.6016,Y -51.4263,Z 98,A -36.5587,B 24.9352,C -1.8598,E1 25.1354,E2 121.9533} C_DIS
Enddeposition()
END
